(* IEC 61131-3 sources: SmartHomeNew/snapshots/2026-05-19 (part 2) *)

(* ---- GVL_STATE.gvl ---- *)
{attribute 'qualified_only'}
VAR_GLOBAL
    G_Floor_Temps : ARRAY[1..GVL_CONSTANTS.C_MAX_HEATING_CIRCUITS] OF REAL;
    G_Room_Temps : ARRAY[1..GVL_CONSTANTS.C_MAX_ZONES] OF REAL;
    G_Last_Valid_Room_Temps : ARRAY[1..GVL_CONSTANTS.C_MAX_ZONES] OF REAL;
    G_Last_Valid_Floor_Temps : ARRAY[1..GVL_CONSTANTS.C_MAX_HEATING_CIRCUITS] OF REAL;
    G_Temp_Sensor_Fault : ARRAY[1..GVL_CONSTANTS.C_MAX_ZONES] OF BOOL;
    G_Floor_Temp_Sensor_Fault : ARRAY[1..GVL_CONSTANTS.C_MAX_HEATING_CIRCUITS] OF BOOL;
    G_Room_Hum : ARRAY[1..GVL_CONSTANTS.C_MAX_ZONES] OF REAL;
    G_Room_CO2 : ARRAY[1..GVL_CONSTANTS.C_MAX_ZONES] OF REAL;
    G_Motion_Sensors : ARRAY[1..GVL_CONSTANTS.C_MAX_LIGHT_ZONES] OF BOOL;
    G_Door_Sensors : ARRAY[1..GVL_CONSTANTS.C_MAX_DOOR_SENSORS] OF BOOL;
    G_Window_Sensors : ARRAY[1..GVL_CONSTANTS.C_MAX_ZONES] OF BOOL;
    G_Water_Sensors : ARRAY[1..GVL_CONSTANTS.C_MAX_FLOOD_SENSORS] OF BOOL;
    G_Flood_Warning : ARRAY[1..GVL_CONSTANTS.C_MAX_FLOOD_SENSORS] OF BOOL;
    G_Flood_Alarm : ARRAY[1..GVL_CONSTANTS.C_MAX_FLOOD_SENSORS] OF BOOL;
    G_Flood_Warning_Rise : ARRAY[1..GVL_CONSTANTS.C_MAX_FLOOD_SENSORS] OF BOOL;
    G_Flood_Alarm_Rise : ARRAY[1..GVL_CONSTANTS.C_MAX_FLOOD_SENSORS] OF BOOL;
    G_Flood_Alarm_Fall : ARRAY[1..GVL_CONSTANTS.C_MAX_FLOOD_SENSORS] OF BOOL;
    G_Smoke_Sensors : ARRAY[1..GVL_CONSTANTS.C_MAX_SMOKE_SENSORS] OF BOOL;
    G_Methane_Sensors : ARRAY[1..GVL_CONSTANTS.C_MAX_METHANE_SENSORS] OF REAL;
    G_CO_Sensors : ARRAY[1..GVL_CONSTANTS.C_MAX_CO_SENSORS] OF REAL;
    G_Manifold_Pressures : ARRAY[1..GVL_CONSTANTS.C_MAX_MANIFOLDS] OF REAL;
    G_Manifold_Currents : ARRAY[1..GVL_CONSTANTS.C_MAX_MANIFOLDS] OF REAL;
    G_Predictive_Pump_Pressure_Drop : ARRAY[1..GVL_CONSTANTS.C_MAX_MANIFOLDS] OF BOOL;
    G_Predictive_Pump_Current_Rise : ARRAY[1..GVL_CONSTANTS.C_MAX_MANIFOLDS] OF BOOL;
    G_Manifold_T_Supply : ARRAY[1..GVL_CONSTANTS.C_MAX_MANIFOLDS] OF REAL;
    G_Manifold_T_Return : ARRAY[1..GVL_CONSTANTS.C_MAX_MANIFOLDS] OF REAL;
    G_Boiler_Flame : ARRAY[1..GVL_CONSTANTS.C_MAX_BOILERS] OF BOOL;
    G_Boiler_Error : ARRAY[1..GVL_CONSTANTS.C_MAX_BOILERS] OF BOOL;
    G_Boiler_OT_Online : ARRAY[1..GVL_CONSTANTS.C_MAX_BOILERS] OF BOOL;
    G_Boiler_OT_Command_Ack : ARRAY[1..GVL_CONSTANTS.C_MAX_BOILERS] OF BOOL;
    G_Boiler_OT_Command_Timeout : ARRAY[1..GVL_CONSTANTS.C_MAX_BOILERS] OF BOOL;
    G_Boiler_OT_Heartbeat_Timeout : ARRAY[1..GVL_CONSTANTS.C_MAX_BOILERS] OF BOOL;
    G_Boiler_OT_Adapter_Error : ARRAY[1..GVL_CONSTANTS.C_MAX_BOILERS] OF BOOL;
    G_Boiler_OT_Heartbeat_Age_MS : ARRAY[1..GVL_CONSTANTS.C_MAX_BOILERS] OF UDINT;
    G_Boiler_OT_Command_Age_MS : ARRAY[1..GVL_CONSTANTS.C_MAX_BOILERS] OF UDINT;
    G_Boiler_OT_Adapter_State : ARRAY[1..GVL_CONSTANTS.C_MAX_BOILERS] OF E_OpenTherm_Adapter_State;
    G_Boiler_OT_Error_State : ARRAY[1..GVL_CONSTANTS.C_MAX_BOILERS] OF E_OpenTherm_Error;
    G_Boiler_OT_Enable : ARRAY[1..GVL_CONSTANTS.C_MAX_BOILERS] OF BOOL;
    G_Boiler_OT_Setpoint : ARRAY[1..GVL_CONSTANTS.C_MAX_BOILERS] OF REAL;
    G_Heating_Cascade_Available : BOOL;
    G_Heating_Cascade_Degraded : BOOL;
    G_Heating_Cascade_Partial_Capacity : BOOL;
    G_Heating_Cascade_No_Flame : BOOL;
    G_Heating_Cascade_Transport_Degraded : BOOL;
    G_Heating_Cascade_Ignition_Timeout : BOOL;
    G_Heating_Cascade_Active_Boilers : UINT;
    G_Heating_Cascade_Available_Boilers : UINT;
    G_Physical_Switches : ARRAY[1..GVL_CONSTANTS.C_MAX_LIGHT_ZONES] OF BOOL;
    G_Socket_Switches : ARRAY[1..GVL_CONSTANTS.C_MAX_SOCKETS] OF BOOL;
    G_Outdoor_Temp : REAL;
    G_Supply_Temps : ARRAY[1..GVL_CONSTANTS.C_MAX_SUPPLY_TEMPS] OF REAL;
    G_DHW_Temp : REAL;
    G_DHW_Pressure : REAL;
    G_Zone_Valves : ARRAY[1..GVL_CONSTANTS.C_MAX_HEATING_CIRCUITS] OF BOOL;
    G_Manifold_Pumps : ARRAY[1..GVL_CONSTANTS.C_MAX_MANIFOLDS] OF BOOL;
    G_Manifold_Valves : ARRAY[1..GVL_CONSTANTS.C_MAX_MANIFOLDS] OF REAL;
    G_Manifold_End_Switches : ARRAY[1..GVL_CONSTANTS.C_MAX_MANIFOLDS] OF BOOL;
    G_Supply_Fans : ARRAY[1..GVL_CONSTANTS.C_MAX_SUPPLY_FANS] OF REAL;
    G_Exhaust_Fans : ARRAY[1..GVL_CONSTANTS.C_MAX_EXHAUST_FANS] OF REAL;
    G_Vent_Heater_Power : ARRAY[1..GVL_CONSTANTS.C_MAX_BOILERS] OF REAL;
    G_Lighting_Levels : ARRAY[1..GVL_CONSTANTS.C_MAX_LIGHT_ZONES] OF BYTE;
    G_Blinds_Positions : ARRAY[1..GVL_CONSTANTS.C_MAX_BLINDS] OF BYTE;
    G_Socket_States : ARRAY[1..GVL_CONSTANTS.C_MAX_SOCKETS] OF BOOL;
    G_DHW_Heating_Pump : BOOL;
    G_DHW_Circ_Pump : BOOL;
    G_Backup_Circulation_Pump : BOOL;
    G_Electric_Heater_Enable : BOOL;
    G_Safety_Gas_Alarm : BOOL;
    G_Safety_Leak_Alarm : BOOL;
    G_Safety_Smoke_Alarm : BOOL;
    G_Safety_Emergency_Stop : BOOL;
    G_Safety_Gas_Latched : BOOL;
    G_Safety_Leak_Latched : BOOL;
    G_Safety_Smoke_Latched : BOOL;
    G_Safety_Freeze_Risk : BOOL;
    G_System_Mode : E_System_Operating_Mode := E_System_Operating_Mode.MODE_NORMAL;
    G_System_Mode_Text : STRING(64);
    G_Heating_IO_Fault : BOOL;
    G_Heating_Sensor_Fault : BOOL;
    G_Heating_Subsystem_Degraded : BOOL;
    G_Allocation_Policy_Active : BOOL;
    G_Allocation_Freeze_Bypass_Active : BOOL;
    G_Allocation_DHW_Bypass_Active : BOOL;
    G_Allocation_Budget_Max : REAL;
    G_Allocation_Budget_Used : REAL;
    G_Allocation_Requested : ARRAY[1..GVL_CONSTANTS.C_MAX_MANIFOLDS] OF BOOL;
    G_Allocation_Allowed : ARRAY[1..GVL_CONSTANTS.C_MAX_MANIFOLDS] OF BOOL;
    G_Allocation_Filtered : ARRAY[1..GVL_CONSTANTS.C_MAX_MANIFOLDS] OF BOOL;
    G_Allocation_Block_Reason : ARRAY[1..GVL_CONSTANTS.C_MAX_MANIFOLDS] OF E_Heating_Allocation_Block_Reason;
    G_Allocation_Effective_Priority : ARRAY[1..GVL_CONSTANTS.C_MAX_MANIFOLDS] OF INT;
    G_Policy_Target_Adjustment_Active : BOOL;
    G_Policy_Target_Adjustment_Applied : REAL;
    G_Policy_Priority_Multiplier_Applied : REAL;
    G_Policy_Priority_Bridge_Active : BOOL;
    G_Policy_Priority_Bias_Applied : ARRAY[1..GVL_CONSTANTS.C_MAX_MANIFOLDS] OF REAL;
    G_Policy_Priority_Effective : ARRAY[1..GVL_CONSTANTS.C_MAX_MANIFOLDS] OF INT;
    G_Heating_RootCause : E_Heating_RootCause := E_Heating_RootCause.RC_NONE;
    G_Heating_RootConfidence : REAL;
    G_Heating_Confidence : REAL := 1.0;
    G_Heating_Error_Score : REAL := 0.0;
    G_Heating_Confidence_Reason_Code : INT := 0;
    G_Heating_Confidence_Reason_Text : STRING(128) := 'OK';
    G_DHW_IO_Fault : BOOL;
    G_DHW_Sensor_Fault : BOOL;
    G_DHW_Subsystem_Degraded : BOOL;
    G_Ventilation_IO_Fault : BOOL;
    G_Ventilation_Subsystem_Degraded : BOOL;
    G_Lighting_IO_Fault : BOOL;
    G_Lighting_Subsystem_Degraded : BOOL;
    G_Access_Comm_Fault : BOOL;
    G_Evacuation_Lighting_Active : BOOL;
    G_Evac_Hazard_Zone : ARRAY[1..GVL_CONSTANTS.C_MAX_LIGHT_ZONES] OF BOOL;
    G_Evac_Guidance : ARRAY[1..GVL_CONSTANTS.C_MAX_LIGHT_ZONES] OF INT;
    G_Rule_Actions : ARRAY[1..GVL_CONSTANTS.C_MAX_RULES] OF ST_Rule_Action;
    G_Sim_Lights : ARRAY[1..GVL_CONSTANTS.C_MAX_LIGHT_ZONES] OF BOOL;
    G_Freeze_Hardware_Degraded : BOOL;
    G_Freeze_Hardware_Failed : BOOL;
    G_Water_Zone_Enable : ARRAY[1..GVL_CONSTANTS.C_MAX_WATER_ZONES] OF BOOL;
    G_Water_Zone_Open_FB : ARRAY[1..GVL_CONSTANTS.C_MAX_WATER_ZONES] OF BOOL;
    G_Water_Zone_Close_FB : ARRAY[1..GVL_CONSTANTS.C_MAX_WATER_ZONES] OF BOOL;
    G_Water_Zone_Exercise_Active : ARRAY[1..GVL_CONSTANTS.C_MAX_WATER_ZONES] OF BOOL;
    G_Preheat_Request : BOOL;
    G_Freeze_Request : BOOL;
    G_Target_Temperature : REAL;
END_VAR

(* ---- GVL_SYSTEM_COORDINATION.gvl ---- *)
{attribute 'qualified_only'}
VAR_GLOBAL
    G_System_Degraded : BOOL := FALSE;

    G_Block_Heating : BOOL := FALSE;
    G_Block_Ventilation : BOOL := FALSE;
    G_Block_Lighting_Override : BOOL := FALSE;
    G_Block_Sockets_Override : BOOL := FALSE;

    G_Coordination_Code : UDINT := 0;
    G_Coordination_Status_Msg : STRING(200) := '';
END_VAR

(* ---- GVL_TEMPORAL_CAUSALITY_CLOSURE_FABRIC.gvl ---- *)
VAR_GLOBAL
    Temporal_Causality_Closure_Valid : BOOL := FALSE;
    Temporal_Causality_Closure_Granted : BOOL := FALSE;

    Temporal_Causality_Coherent : BOOL := FALSE;
    Monotonic_Reality_Timeline_Valid : BOOL := FALSE;
    Distributed_Temporal_Alignment_Stable : BOOL := FALSE;
    Recovery_Revocation_Ordering_Valid : BOOL := FALSE;

    Temporal_Causality_Lineage_Coherent : BOOL := FALSE;
    Distributed_Temporal_Consensus_Valid : BOOL := FALSE;

    Temporal_Fork_Detected : BOOL := FALSE;
    Stale_Causality_Application_Detected : BOOL := FALSE;
    Recovery_Before_Revocation_Detected : BOOL := FALSE;
    Distributed_Timeline_Drift_Detected : BOOL := FALSE;

    Temporal_Causality_Epoch : UDINT := 0;
END_VAR

(* ---- GVL_TEST_PANEL_RESULT.gvl ---- *)
{attribute 'qualified_only'}
VAR_GLOBAL
    // === RESULT VIEW ONLY ===
    G_Enable : BOOL := FALSE;
    G_Scenario_ID : INT := 0;
    G_Scenario_Run : BOOL := FALSE;
    G_Scenario_Active : BOOL := FALSE;

    G_Test_Result_Line : STRING(200) := 'Idle';
    G_Result_Passed : BOOL := FALSE;
    G_Result_Status_Msg : STRING(200) := 'Idle';
    G_Result_Fail_Code : UDINT := 0;

    G_Result_Base_Priority : INT := 0;
    G_Result_Expected_Adjusted_Priority : INT := 0;
    G_Result_Actual_Adjusted_Priority : INT := 0;
    G_Result_Delta : INT := 0;

    G_Result_Budget_Exceeded : BOOL := FALSE;
    G_Result_Used_Thermal_Budget : REAL := 0.0;
    G_Result_Manifold_Enabled : ARRAY[1..GVL_CONSTANTS.C_MAX_MANIFOLDS] OF BOOL;
END_VAR

(* ---- GVL_Water_Isolation_Authority.gvl ---- *)
{attribute 'qualified_only'}
VAR_GLOBAL
    // ==============================================================================
    // Water/Flood authority arbitration publication.
    // ==============================================================================
    //
    // Explicit deterministic authority decision layer.
    //
    // This layer:
    // - evaluates selective isolation authority;
    // - preserves conservative global fallback;
    // - publishes explainable authority decisions.
    //
    // This layer does NOT directly own physical outputs.
    // ==============================================================================

    G_Authority_State : ARRAY[1..GVL_CONSTANTS.C_MAX_FLOOD_SENSORS] OF ST_Water_Isolation_Authority_State;

    // Aggregated authority visibility.
    G_Any_Selective_Authority_Allowed : BOOL;
    G_Any_Global_Fallback_Required : BOOL;
    G_Any_Authority_Denied : BOOL;

    // Runtime lifecycle.
    G_Authority_Valid : BOOL;
    G_Last_Update_MS : UDINT;

    // Explainability.
    G_Status_Code : UINT;
    G_Status_Text : STRING(128);
END_VAR

(* ---- GVL_Water_Output_Reconciliation.gvl ---- *)
{attribute 'qualified_only'}
VAR_GLOBAL
    G_Reconciliation_State : ARRAY[1..64] OF ST_Water_Output_Reconciliation_State;

    G_Any_Runtime_Mismatch : BOOL;
    G_Any_Confirmation_Mismatch : BOOL;
    G_Any_Conflict_Detected : BOOL;

    G_Runtime_Valid : BOOL;
    G_Last_Update_MS : UDINT;

    G_Status_Code : UINT;
    G_Status_Text : STRING(128);
END_VAR

(* ---- GVL_Water_Recovery_Runtime.gvl ---- *)
{attribute 'qualified_only'}
VAR_GLOBAL
    G_Recovery_State : ARRAY[1..64] OF ST_Water_Recovery_Runtime_State;

    G_Any_Recovery_Denied : BOOL;
    G_Any_Unsafe_Recovery : BOOL;

    G_Runtime_Valid : BOOL;
    G_Last_Update_MS : UDINT;

    G_Status_Code : UINT;
    G_Status_Text : STRING(128);
END_VAR

(* ---- GVL_Water_Runtime_Projection.gvl ---- *)
{attribute 'qualified_only'}
VAR_GLOBAL
    // ==============================================================================
    // Canonical Water/Flood runtime projection publication surface.
    // ==============================================================================
    //
    // Observe/publish-only semantic boundary.
    //
    // This GVL is intended to become the canonical semantic transfer layer
    // between:
    //
    // - leak detection/runtime execution;
    // - safety governance;
    // - future selective isolation semantics;
    // - observability/explainability;
    // - supervisory publication.
    //
    // This GVL does NOT:
    // - own outputs;
    // - own valve authority;
    // - directly close/open valves;
    // - override runtime.
    //
    // Canonical topology direction:
    //
    // physical input
    //   -> normalized leak semantics
    //   -> logical leak sensor
    //   -> hydraulic mapping
    //   -> isolation semantics
    //   -> governance/arbitration
    //   -> output projection
    //   -> observability/publication
    // ==============================================================================

    G_Leak_Runtime_State : ARRAY[1..GVL_CONSTANTS.C_MAX_FLOOD_SENSORS] OF ST_Water_Leak_Runtime_State;

    // Projection lifecycle.
    G_Projection_Valid : BOOL;
    G_Last_Projection_MS : UDINT;

    // Active runtime compatibility visibility.
    G_Global_Leak_Active : BOOL;
    G_Global_Warning_Active : BOOL;

    // Observability contract.
    G_Runtime_Projection_Status_Code : UINT;
    G_Runtime_Projection_Status_Text : STRING(128);
END_VAR

(* ---- GVL_Water_Topology_Validation.gvl ---- *)
{attribute 'qualified_only'}
VAR_GLOBAL
    G_Validation_State : ARRAY[1..64] OF ST_Water_Topology_Validation_State;

    G_Any_Invalid : BOOL;
    G_Any_Ambiguous : BOOL;
    G_Any_Global_Fallback_Required : BOOL;

    G_Runtime_Valid : BOOL;
    G_Last_Update_MS : UDINT;

    G_Status_Code : UINT;
    G_Status_Text : STRING(128);
END_VAR

(* ---- GVL_Water_Valve_Feedback.gvl ---- *)
{attribute 'qualified_only'}
VAR_GLOBAL
    G_Valve_Feedback_State : ARRAY[1..64] OF ST_Water_Valve_Feedback_State;

    G_Any_Degraded : BOOL;
    G_Any_Timeout : BOOL;
    G_Any_Conflict : BOOL;

    G_Runtime_Valid : BOOL;
    G_Last_Update_MS : UDINT;

    G_Status_Code : UINT;
    G_Status_Text : STRING(128);
END_VAR

(* ---- FB_Access_Output_Projection.st ---- *)
FUNCTION_BLOCK FB_Access_Output_Projection
VAR_INPUT
    VI_Lock_1_Open : BOOL;
    VI_Lock_1_Close : BOOL;
    VI_Lock_2_Open : BOOL;
    VI_Lock_2_Close : BOOL;
    VI_Gate_Open : BOOL;
    VI_Wicket_Open : BOOL;
END_VAR

GVL_ACCESS_OUTPUT.DO_Lock_1_Open := VI_Lock_1_Open;
GVL_ACCESS_OUTPUT.DO_Lock_1_Close := VI_Lock_1_Close;
GVL_ACCESS_OUTPUT.DO_Lock_2_Open := VI_Lock_2_Open;
GVL_ACCESS_OUTPUT.DO_Lock_2_Close := VI_Lock_2_Close;
GVL_ACCESS_OUTPUT.DO_Gate_Open := VI_Gate_Open;
GVL_ACCESS_OUTPUT.DO_Wicket_Open := VI_Wicket_Open;

END_FUNCTION_BLOCK
// >>> BULK_SYNC_ANCHOR: FB_Access_Output_Projection <<<

(* ---- FB_ADS_Runtime_Adapter.st ---- *)
FUNCTION_BLOCK FB_ADS_Runtime_Adapter
VAR_INPUT
    VI_Enable : BOOL;
    VI_System_Time_MS : UDINT;
END_VAR
VAR
    L_Frame : ST_Runtime_Bus_Frame;
    L_TX_Index : UINT;
END_VAR

IF NOT VI_Enable THEN
    RETURN;
END_IF;

L_TX_Index := UDINT_TO_UINT(GVL_Runtime_Bus.G_Last_Sequence_Id);

IF (L_TX_Index >= 1)
   AND (L_TX_Index <= 128) THEN

    L_Frame := GVL_Runtime_Bus.G_TX_Frames[L_TX_Index];

    IF L_Frame.Frame_Valid THEN

        IF GVL_Distributed_Authority.G_Distributed_Safety_Barrier_OK
           AND GVL_Runtime_Sessions.G_Runtime_Valid
           AND NOT GVL_Runtime_Sessions.G_Any_Stale_Session
           AND NOT GVL_Runtime_Sessions.G_Any_Quarantined_Session THEN

            L_Frame.Frame_Ack_Received := TRUE;
            L_Frame.Replication_Consistent := TRUE;
            L_Frame.Replication_Rejected := FALSE;
            L_Frame.Status_Code := 0;

        ELSE

            L_Frame.Frame_Ack_Received := FALSE;
            L_Frame.Replication_Consistent := FALSE;
            L_Frame.Replication_Rejected := TRUE;
            L_Frame.Status_Code := 2;

        END_IF;

        GVL_Runtime_Bus.G_TX_Frames[L_TX_Index] := L_Frame;
        GVL_Runtime_Bus.G_TX_Healthy := L_Frame.Replication_Consistent;
        GVL_Runtime_Bus.G_Any_Replication_Rejected := L_Frame.Replication_Rejected;

    END_IF;

END_IF;

END_FUNCTION_BLOCK

(* ---- FB_Behavior_Adapt.st ---- *)
FUNCTION_BLOCK FB_Behavior_Adapt
VAR_INPUT
    iScenario : E_System_Reason_Code;
    iSuccess : BOOL;
    iMeasuredValue : REAL;
    iZone : INT;
    iConfidence : REAL;
END_VAR

VAR
    L_Stats : ST_Scenario_Stats;
    L_Zone : ST_Zone_Adapt_State;
    L_Adjustment : REAL;
    L_Decay : REAL;
    idx : INT;
END_VAR

IF NOT GVL_BEHAVIOR_ADAPT.G_Adapt_Enabled THEN RETURN; END_IF;

idx := USINT_TO_INT(iScenario);

L_Stats := GVL_BEHAVIOR_ADAPT.G_Scenario_Stats[idx];
L_Stats.Activations := L_Stats.Activations + 1;

IF iSuccess THEN
    L_Stats.Success_Count := L_Stats.Success_Count + 1;
ELSE
    L_Stats.Failure_Count := L_Stats.Failure_Count + 1;
END_IF;

IF L_Stats.Activations > 0 THEN
    L_Stats.Success_Rate := UDINT_TO_REAL(L_Stats.Success_Count) / UDINT_TO_REAL(L_Stats.Activations);
END_IF;

IF (iScenario = REASON_SCENARIO_VENT_BOOST) AND (iZone >= 1) AND (iZone <= GVL_CONSTANTS.C_MAX_ZONES) THEN

    L_Zone := GVL_BEHAVIOR_ADAPT.G_VentBoost_Zone_Adapt[iZone];

    IF L_Zone.Zone_Weight = 0.0 THEN
        L_Zone.Zone_Weight := GVL_BEHAVIOR_ADAPT.G_Adapt_Default_Zone_Weight;
    END_IF;

    L_Decay := GVL_BEHAVIOR_ADAPT.G_Decay_Factor;
    L_Zone.Zone_Weight := L_Zone.Zone_Weight * L_Decay;
    L_Zone.Confidence := L_Zone.Confidence * L_Decay;

    L_Zone.Activations := L_Zone.Activations + 1;

    IF iSuccess THEN
        L_Zone.Success_Count := L_Zone.Success_Count + 1;
    ELSE
        L_Zone.Failure_Count := L_Zone.Failure_Count + 1;
    END_IF;

    IF L_Zone.Activations > 0 THEN
        L_Zone.Success_Rate := UDINT_TO_REAL(L_Zone.Success_Count) / UDINT_TO_REAL(L_Zone.Activations);
    END_IF;

    IF iConfidence >= GVL_BEHAVIOR_ADAPT.G_Adapt_Min_Confidence THEN
        L_Zone.Confidence := L_Zone.Confidence +
            (iConfidence - L_Zone.Confidence) * GVL_BEHAVIOR_ADAPT.G_Confidence_Learning_Rate;
    END_IF;

    IF (GVL_BEHAVIOR_ADAPT.G_Adapt_Update_Threshold > 0) AND
       ((L_Zone.Activations MOD INT_TO_UDINT(GVL_BEHAVIOR_ADAPT.G_Adapt_Update_Threshold)) = 0) THEN

        L_Adjustment :=
            (L_Zone.Success_Rate - 0.5)
            * GVL_BEHAVIOR_ADAPT.G_Adapt_Learning_Rate
            * L_Zone.Confidence;

        L_Zone.Zone_Weight := LIMIT(0.5, L_Zone.Zone_Weight + L_Adjustment, 2.0);

    END_IF;

    L_Zone.Last_Update_MS := GVL_TIME_SERVICE.G_Now_MS;

    GVL_BEHAVIOR_ADAPT.G_VentBoost_Zone_Adapt[iZone] := L_Zone;

END_IF;

GVL_BEHAVIOR_ADAPT.G_Scenario_Stats[idx] := L_Stats;
END_FUNCTION_BLOCK

(* ---- FB_Boiler_Cascade_Manager.st ---- *)
FUNCTION_BLOCK FB_Boiler_Cascade_Manager
VAR_INPUT
    VI_Enable : BOOL;
    VI_System_Time_MS : UDINT;
    VI_Boiler_Stop : BOOL;

    VI_DHW_Heating_Demand : BOOL;
    VI_DHW_Target_Temp : REAL;

    VI_Target_Supply_Temp : REAL;
    VI_Demand_Power : REAL; // 0..500% (сумма запросов от 5 смесительных узлов)

    VI_Boiler_Flame_Status : ARRAY[1..GVL_CONSTANTS.C_MAX_BOILERS] OF BOOL;
    VI_Boiler_Error_Status : ARRAY[1..GVL_CONSTANTS.C_MAX_BOILERS] OF BOOL;
    VI_Boiler_OT_Online : ARRAY[1..GVL_CONSTANTS.C_MAX_BOILERS] OF BOOL;
    VI_Boiler_Modulation : ARRAY[1..GVL_CONSTANTS.C_MAX_BOILERS] OF REAL;
END_VAR

VAR_OUTPUT
    VO_Boiler_Enable : ARRAY[1..GVL_CONSTANTS.C_MAX_BOILERS] OF BOOL;
    VO_Boiler_Setpoint : ARRAY[1..GVL_CONSTANTS.C_MAX_BOILERS] OF REAL;
    VO_Lead_Boiler : BYTE;
END_VAR

VAR
    L_i : INT;
    L_Lead_Boiler : BYTE := 1;

    L_Last_Rotation_MS : UDINT := 0;
    L_Rotation_Initialized : BOOL := FALSE;
    L_Rotation_Period_MS : UDINT := 604800000; // 168h

    L_Lead_Available : BOOL;
    L_Reserve_Available : BOOL;
    L_Reserve_Boiler : BYTE;
    L_Start_Reserve : BOOL;
    L_Target_Setpoint : REAL;
    L_Flame_Miss_Timer : ARRAY[1..GVL_CONSTANTS.C_MAX_BOILERS] OF TON;
END_VAR

// Сброс выходов по умолчанию
FOR L_i := 1 TO GVL_CONSTANTS.C_MAX_BOILERS DO
    VO_Boiler_Enable[L_i] := FALSE;
    VO_Boiler_Setpoint[L_i] := 0.0;
END_FOR;

// Инициализация ротации
IF NOT L_Rotation_Initialized THEN
    L_Last_Rotation_MS := VI_System_Time_MS;
    L_Rotation_Initialized := TRUE;
END_IF;

// Принудительная остановка
IF VI_Boiler_Stop THEN
    VO_Lead_Boiler := L_Lead_Boiler;
    RETURN;
END_IF;

// Ротация строго каждые 168 часов
IF (VI_System_Time_MS - L_Last_Rotation_MS) >= L_Rotation_Period_MS THEN
    IF GVL_CONSTANTS.C_MAX_BOILERS > 1 THEN
        L_Lead_Boiler := 3 - L_Lead_Boiler;
    END_IF;
    L_Last_Rotation_MS := VI_System_Time_MS;
END_IF;

L_Reserve_Boiler := SEL(L_Lead_Boiler = 1, 1, 2);

L_Lead_Available :=
    VI_Boiler_OT_Online[L_Lead_Boiler] AND
    NOT VI_Boiler_Error_Status[L_Lead_Boiler];

L_Reserve_Available :=
    (GVL_CONSTANTS.C_MAX_BOILERS > 1) AND
    VI_Boiler_OT_Online[L_Reserve_Boiler] AND
    NOT VI_Boiler_Error_Status[L_Reserve_Boiler];

// Контроль "команда есть, пламени нет" для ведущего котла
L_Flame_Miss_Timer[L_Lead_Boiler](
    IN := VI_Enable AND L_Lead_Available AND NOT VI_DHW_Heating_Demand AND NOT VI_Boiler_Flame_Status[L_Lead_Boiler],
    PT := T#120s
);

IF L_Flame_Miss_Timer[L_Lead_Boiler].Q AND L_Reserve_Available THEN
    L_Lead_Boiler := L_Reserve_Boiler;
    L_Last_Rotation_MS := VI_System_Time_MS;
    L_Lead_Available :=
        VI_Boiler_OT_Online[L_Lead_Boiler] AND
        NOT VI_Boiler_Error_Status[L_Lead_Boiler];
    L_Reserve_Boiler := SEL(L_Lead_Boiler = 1, 1, 2);
    L_Reserve_Available :=
        (GVL_CONSTANTS.C_MAX_BOILERS > 1) AND
        VI_Boiler_OT_Online[L_Reserve_Boiler] AND
        NOT VI_Boiler_Error_Status[L_Reserve_Boiler];
END_IF;

// Нет запроса тепла
IF NOT VI_Enable THEN
    VO_Lead_Boiler := L_Lead_Boiler;
    RETURN;
END_IF;

// Целевая уставка
IF VI_DHW_Heating_Demand THEN
    L_Target_Setpoint := LIMIT(20.0, VI_DHW_Target_Temp + 15.0, 85.0);
ELSE
    L_Target_Setpoint := LIMIT(20.0, VI_Target_Supply_Temp + 5.0, 80.0);
END_IF;

// Выбор ведущего по доступности
IF NOT L_Lead_Available AND L_Reserve_Available THEN
    L_Lead_Boiler := L_Reserve_Boiler;
    L_Lead_Available := TRUE;
    L_Reserve_Boiler := SEL(L_Lead_Boiler = 1, 1, 2);
    L_Reserve_Available :=
        (GVL_CONSTANTS.C_MAX_BOILERS > 1) AND
        VI_Boiler_OT_Online[L_Reserve_Boiler] AND
        NOT VI_Boiler_Error_Status[L_Reserve_Boiler];
END_IF;

// Основной котёл
IF L_Lead_Available THEN
    VO_Boiler_Enable[L_Lead_Boiler] := TRUE;
    VO_Boiler_Setpoint[L_Lead_Boiler] := L_Target_Setpoint;
END_IF;

// Резервный котёл: >80% или отказ основного
L_Start_Reserve :=
    L_Reserve_Available AND
    (
        (VI_Demand_Power > 80.0) OR
        (NOT L_Lead_Available)
    );

IF L_Start_Reserve THEN
    VO_Boiler_Enable[L_Reserve_Boiler] := TRUE;
    VO_Boiler_Setpoint[L_Reserve_Boiler] := L_Target_Setpoint;
END_IF;

VO_Lead_Boiler := L_Lead_Boiler;
END_FUNCTION_BLOCK

(* ---- FB_Boiler_OpenTherm_Interface.st ---- *)
FUNCTION_BLOCK FB_Boiler_OpenTherm_Interface
VAR_INPUT
    VI_Enable : ARRAY[1..GVL_CONSTANTS.C_MAX_BOILERS] OF BOOL;
    VI_Setpoint : ARRAY[1..GVL_CONSTANTS.C_MAX_BOILERS] OF REAL;

    VI_OT_Online : ARRAY[1..GVL_CONSTANTS.C_MAX_BOILERS] OF BOOL;
    VI_OT_Error : ARRAY[1..GVL_CONSTANTS.C_MAX_BOILERS] OF BOOL;
END_VAR

VAR_OUTPUT
    VO_OT_Enable : ARRAY[1..GVL_CONSTANTS.C_MAX_BOILERS] OF BOOL;
    VO_OT_Setpoint : ARRAY[1..GVL_CONSTANTS.C_MAX_BOILERS] OF REAL;
    VO_OT_Command_Valid : ARRAY[1..GVL_CONSTANTS.C_MAX_BOILERS] OF BOOL;
END_VAR

VAR
    L_i : INT;
    L_Setpoint : REAL;
    L_Setpoint_x10 : UINT;
    L_Command_Enable : BOOL;
    L_Command_Changed : BOOL;
    L_Last_Command_Enable : ARRAY[1..GVL_CONSTANTS.C_MAX_BOILERS] OF BOOL;
    L_Last_Command_Setpoint_x10 : ARRAY[1..GVL_CONSTANTS.C_MAX_BOILERS] OF UINT;
END_VAR

FOR L_i := 1 TO GVL_CONSTANTS.C_MAX_BOILERS DO

    VO_OT_Enable[L_i] := FALSE;
    VO_OT_Setpoint[L_i] := 0.0;
    VO_OT_Command_Valid[L_i] := FALSE;

    L_Command_Enable := FALSE;
    L_Setpoint := 0.0;
    L_Setpoint_x10 := 0;

    // ======================================================
    // COMMAND VALIDATION
    // ======================================================
    IF VI_Enable[L_i] AND VI_OT_Online[L_i] AND NOT VI_OT_Error[L_i] THEN
        L_Command_Enable := TRUE;
        L_Setpoint := LIMIT(20.0, VI_Setpoint[L_i], 80.0);
        L_Setpoint_x10 := REAL_TO_UINT(L_Setpoint * 10.0);

        VO_OT_Enable[L_i] := TRUE;
        VO_OT_Setpoint[L_i] := L_Setpoint;
    END_IF;

    // ======================================================
    // PHYSICAL ADAPTER COMMAND IMAGE
    // ======================================================
    GVL_OPENTHERM_ADAPTER.G_Command[L_i].Enable := L_Command_Enable;
    GVL_OPENTHERM_ADAPTER.G_Command[L_i].Setpoint_x10 := L_Setpoint_x10;

    // Sequence is advanced only when the actual command image changes.
    // This keeps the command stable long enough for adapter ACK validation.
    L_Command_Changed :=
        (L_Command_Enable <> L_Last_Command_Enable[L_i]) OR
        (L_Setpoint_x10 <> L_Last_Command_Setpoint_x10[L_i]);

    IF L_Command_Changed THEN
        GVL_OPENTHERM_ADAPTER.G_Command[L_i].Sequence :=
            GVL_OPENTHERM_ADAPTER.G_Command[L_i].Sequence + 1;

        GVL_OPENTHERM_ADAPTER.G_Command[L_i].Last_Write_MS :=
            GVL_STATUS.G_System_Time_MS;

        L_Last_Command_Enable[L_i] := L_Command_Enable;
        L_Last_Command_Setpoint_x10[L_i] := L_Setpoint_x10;
    END_IF;

    // Command is valid only when the adapter confirms the current stable sequence.
    VO_OT_Command_Valid[L_i] :=
        L_Command_Enable AND
        GVL_OPENTHERM_ADAPTER.G_Status[L_i].Command_Ack AND
        (NOT GVL_OPENTHERM_ADAPTER.G_Status[L_i].Adapter_Error) AND
        GVL_OPENTHERM_ADAPTER.G_Status[L_i].Adapter_Online;

END_FOR;

END_FUNCTION_BLOCK

(* ---- FB_Cluster_Runtime_FSM.st ---- *)
FUNCTION_BLOCK FB_Cluster_Runtime_FSM
VAR_INPUT
    VI_Enable : BOOL;
    VI_System_Time_MS : UDINT;
END_VAR
VAR
    L_Finalized_Runtime_Continuity : BOOL;
END_VAR

IF NOT VI_Enable THEN
    GVL_Cluster_Runtime_FSM.G_Runtime_Valid := FALSE;
    RETURN;
END_IF;

// Finalized runtime continuity proof chain.
L_Finalized_Runtime_Continuity :=
    GVL_SEMANTIC_PROGRESS.Semantic_Forward_Progress_Valid
    AND GVL_SEMANTIC_PROGRESS.Semantic_Execution_Continuity_OK
    AND NOT GVL_SEMANTIC_PROGRESS.Semantic_Progress_Lease_Expired
    AND NOT GVL_SEMANTIC_PROGRESS.Semantic_Progress_Quarantine_Active
    AND GVL_RUNTIME_SNAPSHOT.Snapshot_Frozen
    AND GVL_RUNTIME_SNAPSHOT.Snapshot_Publication_Allowed
    AND GVL_RUNTIME_SNAPSHOT.Snapshot_Copy_Valid
    AND GVL_RUNTIME_SNAPSHOT.Snapshot_Isolation_Valid
    AND NOT GVL_RUNTIME_SNAPSHOT.Snapshot_Mutation_Detected
    AND GVL_DISTRIBUTED_SNAPSHOT.Distributed_Publication_Reconciled
    AND GVL_DISTRIBUTED_SNAPSHOT.Distributed_Publication_Freeze_Valid
    AND GVL_DISTRIBUTED_SNAPSHOT.Distributed_Snapshot_Consistent
    AND GVL_DISTRIBUTED_COMMIT.Distributed_Commit_Valid
    AND GVL_DISTRIBUTED_COMMIT.Publication_Prepare_Valid
    AND GVL_DISTRIBUTED_COMMIT.Publication_Commit_Confirmed
    AND NOT GVL_DISTRIBUTED_COMMIT.Peer_Commit_Mismatch
    AND NOT GVL_DISTRIBUTED_COMMIT.Commit_Lease_Expired
    AND GVL_OUTPUT_EPOCH.Output_Publication_Valid
    AND GVL_OUTPUT_EPOCH.Output_Runtime_Epoch_Valid
    AND NOT GVL_OUTPUT_EPOCH.Output_Lease_Expired
    AND NOT GVL_OUTPUT_EPOCH.Output_Forced_Safe_Decay
    AND GVL_COMMAND_VERIFY.PreOutput_Barrier_OK
    AND NOT GVL_COMMAND_VERIFY.PreOutput_Block_IO;

// Reset runtime states.
GVL_Cluster_Runtime_FSM.G_State_Startup := FALSE;
GVL_Cluster_Runtime_FSM.G_State_Discovery := FALSE;
GVL_Cluster_Runtime_FSM.G_State_Synchronization := FALSE;
GVL_Cluster_Runtime_FSM.G_State_Operational := FALSE;
GVL_Cluster_Runtime_FSM.G_State_Degraded := FALSE;
GVL_Cluster_Runtime_FSM.G_State_Observer_Only := FALSE;
GVL_Cluster_Runtime_FSM.G_State_Recovery_Lock := FALSE;
GVL_Cluster_Runtime_FSM.G_State_Quarantine := FALSE;

// Startup state.
IF NOT GVL_Distributed_Runtime.G_Runtime_Valid THEN

    GVL_Cluster_Runtime_FSM.G_State_Startup := TRUE;

    GVL_Cluster_Runtime_FSM.G_Status_Code := 1;
    GVL_Cluster_Runtime_FSM.G_Status_Text :=
        'Cluster runtime startup';

ELSIF GVL_Runtime_Discovery.G_Runtime_Valid
   AND NOT GVL_Runtime_Discovery.G_Any_Discovery_Rejected THEN

    GVL_Cluster_Runtime_FSM.G_State_Discovery := TRUE;

    GVL_Cluster_Runtime_FSM.G_Status_Code := 2;
    GVL_Cluster_Runtime_FSM.G_Status_Text :=
        'Cluster runtime discovery';

END_IF;

// Synchronization state.
IF GVL_Runtime_Bus.G_TX_Healthy
   AND GVL_Runtime_Bus.G_RX_Healthy THEN

    GVL_Cluster_Runtime_FSM.G_State_Synchronization := TRUE;

END_IF;

// Operational state.
IF GVL_Distributed_Execution_Gates.G_Can_Execute
   AND GVL_Distributed_Execution_Gates.G_Can_Orchestrate
   AND L_Finalized_Runtime_Continuity THEN

    GVL_Cluster_Runtime_FSM.G_State_Operational := TRUE;

    GVL_Cluster_Runtime_FSM.G_Status_Code := 0;
    GVL_Cluster_Runtime_FSM.G_Status_Text :=
        'Cluster runtime operational';

END_IF;

// Degraded state.
IF GVL_Cluster_Safety_Barrier.G_Cluster_Execution_Blocked THEN

    GVL_Cluster_Runtime_FSM.G_State_Degraded := TRUE;

    GVL_Cluster_Runtime_FSM.G_Status_Code := 10;
    GVL_Cluster_Runtime_FSM.G_Status_Text :=
        'Cluster runtime degraded';

END_IF;

// Observer-only state.
IF GVL_Distributed_Authority.G_Authority_State.Authority_Observer_Only THEN

    GVL_Cluster_Runtime_FSM.G_State_Observer_Only := TRUE;

    GVL_Cluster_Runtime_FSM.G_Status_Code := 11;
    GVL_Cluster_Runtime_FSM.G_Status_Text :=
        'Cluster runtime observer-only';

END_IF;

// Recovery lock state.
IF GVL_Distributed_Recovery_Lock.G_Recovery_Execution_Blocked THEN

    GVL_Cluster_Runtime_FSM.G_State_Recovery_Lock := TRUE;

    GVL_Cluster_Runtime_FSM.G_Status_Code := 12;
    GVL_Cluster_Runtime_FSM.G_Status_Text :=
        'Cluster runtime recovery-locked';

END_IF;

// Quarantine state.
IF GVL_Runtime_Discovery.G_Any_Node_Quarantined THEN

    GVL_Cluster_Runtime_FSM.G_State_Quarantine := TRUE;

    GVL_Cluster_Runtime_FSM.G_Status_Code := 13;
    GVL_Cluster_Runtime_FSM.G_Status_Text :=
        'Cluster runtime quarantined';

END_IF;

GVL_Cluster_Runtime_FSM.G_Runtime_Valid := TRUE;
GVL_Cluster_Runtime_FSM.G_Last_Update_MS := VI_System_Time_MS;

END_FUNCTION_BLOCK

(* ---- FB_Cluster_Safety_Barrier_Runtime.st ---- *)
FUNCTION_BLOCK FB_Cluster_Safety_Barrier_Runtime
VAR_INPUT
    VI_Enable : BOOL;
    VI_System_Time_MS : UDINT;
END_VAR
VAR
    L_Block_Execution : BOOL;
    L_Status_Code : UINT;
    L_Status_Text : STRING(160);

    L_Finalized_Runtime_Continuity : BOOL;
END_VAR

IF NOT VI_Enable THEN
    GVL_Cluster_Safety_Barrier.G_Runtime_Valid := FALSE;
    RETURN;
END_IF;

L_Block_Execution := FALSE;
L_Status_Code := 0;
L_Status_Text := 'Cluster safety barrier healthy';

GVL_Cluster_Safety_Barrier.G_Remote_Authority_Degraded := FALSE;
GVL_Cluster_Safety_Barrier.G_Runtime_Bus_Degraded := FALSE;
GVL_Cluster_Safety_Barrier.G_Projection_Ownership_Invalid := FALSE;
GVL_Cluster_Safety_Barrier.G_Recovery_Lock_Active := FALSE;
GVL_Cluster_Safety_Barrier.G_Deployment_Invalid := FALSE;
GVL_Cluster_Safety_Barrier.G_Authority_Downgraded := FALSE;
GVL_Cluster_Safety_Barrier.G_Orchestration_Restricted := FALSE;

// Finalized runtime continuity proof chain.
L_Finalized_Runtime_Continuity :=
    GVL_SEMANTIC_PROGRESS.Semantic_Forward_Progress_Valid
    AND GVL_SEMANTIC_PROGRESS.Semantic_Execution_Continuity_OK
    AND NOT GVL_SEMANTIC_PROGRESS.Semantic_Progress_Lease_Expired
    AND NOT GVL_SEMANTIC_PROGRESS.Semantic_Progress_Quarantine_Active
    AND GVL_RUNTIME_SNAPSHOT.Snapshot_Frozen
    AND GVL_RUNTIME_SNAPSHOT.Snapshot_Publication_Allowed
    AND GVL_RUNTIME_SNAPSHOT.Snapshot_Copy_Valid
    AND GVL_RUNTIME_SNAPSHOT.Snapshot_Isolation_Valid
    AND NOT GVL_RUNTIME_SNAPSHOT.Snapshot_Mutation_Detected
    AND GVL_DISTRIBUTED_SNAPSHOT.Distributed_Publication_Reconciled
    AND GVL_DISTRIBUTED_SNAPSHOT.Distributed_Publication_Freeze_Valid
    AND GVL_DISTRIBUTED_SNAPSHOT.Distributed_Snapshot_Consistent
    AND GVL_DISTRIBUTED_COMMIT.Distributed_Commit_Valid
    AND GVL_DISTRIBUTED_COMMIT.Publication_Prepare_Valid
    AND GVL_DISTRIBUTED_COMMIT.Publication_Commit_Confirmed
    AND NOT GVL_DISTRIBUTED_COMMIT.Peer_Commit_Mismatch
    AND NOT GVL_DISTRIBUTED_COMMIT.Commit_Lease_Expired
    AND GVL_OUTPUT_EPOCH.Output_Publication_Valid
    AND GVL_OUTPUT_EPOCH.Output_Runtime_Epoch_Valid
    AND NOT GVL_OUTPUT_EPOCH.Output_Lease_Expired
    AND NOT GVL_OUTPUT_EPOCH.Output_Forced_Safe_Decay
    AND GVL_COMMAND_VERIFY.PreOutput_Barrier_OK
    AND NOT GVL_COMMAND_VERIFY.PreOutput_Block_IO;

// Root finalized continuity barrier.
IF NOT L_Finalized_Runtime_Continuity THEN

    L_Block_Execution := TRUE;
    L_Status_Code := 9;
    L_Status_Text :=
        'Finalized runtime continuity invalid';

    GVL_Cluster_Safety_Barrier.G_Authority_Downgraded := TRUE;
    GVL_Cluster_Safety_Barrier.G_Orchestration_Restricted := TRUE;

END_IF;

// Remote authority staleness barrier.
IF GVL_Distributed_Runtime.G_Any_Remote_Node_Offline
   OR GVL_Distributed_Runtime.G_Split_Brain_Suspected THEN

    L_Block_Execution := TRUE;
    L_Status_Code := 10;
    L_Status_Text :=
        'Cluster authority state degraded';

    GVL_Cluster_Safety_Barrier.G_Remote_Authority_Degraded := TRUE;

END_IF;

// Runtime bus integrity barrier.
IF GVL_Runtime_Bus.G_Any_Replication_Rejected
   OR NOT GVL_Runtime_Bus.G_TX_Healthy
   OR NOT GVL_Runtime_Bus.G_RX_Healthy THEN

    L_Block_Execution := TRUE;
    L_Status_Code := 11;
    L_Status_Text :=
        'Runtime bus integrity degraded';

    GVL_Cluster_Safety_Barrier.G_Runtime_Bus_Degraded := TRUE;

END_IF;

// Projection ownership barrier.
IF GVL_Distributed_Projection_Ownership.G_Any_Ownership_Conflict
   OR GVL_Distributed_Projection_Ownership.G_Any_Ownership_Stale THEN

    L_Block_Execution := TRUE;
    L_Status_Code := 12;
    L_Status_Text :=
        'Distributed projection ownership invalid';

    GVL_Cluster_Safety_Barrier.G_Projection_Ownership_Invalid := TRUE;

END_IF;

// Recovery lock barrier.
IF GVL_Distributed_Recovery_Lock.G_Recovery_Execution_Blocked
   OR GVL_Distributed_Recovery_Lock.G_Rollback_Execution_Blocked
   OR GVL_Distributed_Recovery_Lock.G_Reopen_Execution_Blocked THEN

    L_Block_Execution := TRUE;
    L_Status_Code := 13;
    L_Status_Text :=
        'Distributed recovery execution blocked';

    GVL_Cluster_Safety_Barrier.G_Recovery_Lock_Active := TRUE;

END_IF;

// Discovery/deployment barrier.
IF GVL_Runtime_Discovery.G_Any_Discovery_Rejected
   OR GVL_Runtime_Discovery.G_Any_Node_Quarantined THEN

    L_Block_Execution := TRUE;
    L_Status_Code := 14;
    L_Status_Text :=
        'Runtime deployment/discovery invalid';

    GVL_Cluster_Safety_Barrier.G_Deployment_Invalid := TRUE;

END_IF;

// Cluster escalation semantics.
IF L_Block_Execution THEN

    GVL_Distributed_Authority.G_Authority_State.Authority_Observer_Only := TRUE;
    GVL_Distributed_Authority.G_Authority_State.Authority_Master_Elected := FALSE;

    GVL_Distributed_Orchestration.G_Distributed_Projection_Healthy := FALSE;

    GVL_Cluster_Safety_Barrier.G_Authority_Downgraded := TRUE;
    GVL_Cluster_Safety_Barrier.G_Orchestration_Restricted := TRUE;

END_IF;

GVL_Cluster_Safety_Barrier.G_Cluster_Execution_Blocked :=
    L_Block_Execution;

GVL_Cluster_Safety_Barrier.G_Runtime_Valid := TRUE;
GVL_Cluster_Safety_Barrier.G_Last_Update_MS := VI_System_Time_MS;
GVL_Cluster_Safety_Barrier.G_Status_Code := L_Status_Code;
GVL_Cluster_Safety_Barrier.G_Status_Text := L_Status_Text;

END_FUNCTION_BLOCK

(* ---- FB_Device_Predictive_Diag.st ---- *)
FUNCTION_BLOCK FB_Device_Predictive_Diag
VAR_INPUT
    VI_Current_Value : REAL;      // Текущий ток или время
    VI_Nominal_Value : REAL;      // Эталонное значение
    VI_Is_Running    : BOOL;
    VI_Reset_Stats   : BOOL;
    VI_System_Time_MS: UDINT;     // Системное время (мс)
END_VAR
VAR_IN_OUT
    VIO_Health_Data  : ST_Device_Health;
END_VAR
VAR
    L_Prev_Running   : BOOL;
    L_Start_Time     : UDINT;
    L_Last_Calc_Time : UDINT;
    L_Elapsed_MS     : UDINT;
    L_Accumulated_MS : UDINT; // Накопленное время работы (мс)
    L_Timer_Running  : FB_System_Timer;
END_VAR

// 0. Сброс статистики
IF VI_Reset_Stats THEN
    VIO_Health_Data.Starts_Count := 0;
    VIO_Health_Data.Sample_Count := 0;
    VIO_Health_Data.Current_Sum := 0.0;
    VIO_Health_Data.Avg_Start_Current := 0.0;
    VIO_Health_Data.Health_Score := 100;
    VIO_Health_Data.Maintenance_Required := FALSE;
    VIO_Health_Data.Warning_Message := '';
    VIO_Health_Data.Last_Start_Current := 0.0;
    VIO_Health_Data.Total_Runtime_Hours := 0;
    L_Accumulated_MS := 0;
END_IF;

// 1. Счётчик пусков и замер пускового тока
IF VI_Is_Running AND NOT L_Prev_Running THEN
    VIO_Health_Data.Starts_Count := VIO_Health_Data.Starts_Count + 1;
    VIO_Health_Data.Last_Start_Current := VI_Current_Value;
    L_Start_Time := VI_System_Time_MS;
    L_Last_Calc_Time := VI_System_Time_MS;

    // Обновление среднего пускового тока
    VIO_Health_Data.Sample_Count := VIO_Health_Data.Sample_Count + 1;
    VIO_Health_Data.Current_Sum := VIO_Health_Data.Current_Sum + VI_Current_Value;
    VIO_Health_Data.Avg_Start_Current := VIO_Health_Data.Current_Sum / UDINT_TO_REAL(VIO_Health_Data.Sample_Count);

    // 2. Анализ отклонения пускового тока (п. 12.1 ТЗ)
    IF VI_Current_Value > (VI_Nominal_Value * 1.5) THEN
        VIO_Health_Data.Health_Score := TO_BYTE(LIMIT(0, TO_INT(VIO_Health_Data.Health_Score) - 5, 100));
    ELSIF VI_Current_Value > (VI_Nominal_Value * 1.2) THEN
        VIO_Health_Data.Health_Score := TO_BYTE(LIMIT(0, TO_INT(VIO_Health_Data.Health_Score) - 1, 100));
    ELSIF VI_Current_Value < (VI_Nominal_Value * 0.5) THEN
        VIO_Health_Data.Health_Score := TO_BYTE(LIMIT(0, TO_INT(VIO_Health_Data.Health_Score) - 2, 100));
    END_IF;
END_IF;

// 3. Анализ рабочего тока и наработки
IF VI_Is_Running THEN
    L_Elapsed_MS := (VI_System_Time_MS - L_Last_Calc_Time);
    L_Accumulated_MS := L_Accumulated_MS + L_Elapsed_MS;
    L_Last_Calc_Time := VI_System_Time_MS;

    // Обновляем наработку каждый час (3600000 мс)
    IF L_Accumulated_MS >= 3600000 THEN
        VIO_Health_Data.Total_Runtime_Hours := VIO_Health_Data.Total_Runtime_Hours + 1;
        L_Accumulated_MS := L_Accumulated_MS - 3600000;

        // Естественный износ: -1% здоровья каждые 1000 часов
        IF (VIO_Health_Data.Total_Runtime_Hours MOD 1000) = 0 THEN
            VIO_Health_Data.Health_Score := TO_BYTE(LIMIT(0, TO_INT(VIO_Health_Data.Health_Score) - 1, 100));
        END_IF;

        // Анализ рабочего тока (после пускового режима)
        IF (VI_System_Time_MS - L_Start_Time) > 10000 THEN // 10 секунд после пуска
            IF VI_Current_Value > (VI_Nominal_Value * 1.1) THEN
                // Повышенный рабочий ток - ускоренный износ (-1% в час)
                VIO_Health_Data.Health_Score := TO_BYTE(LIMIT(0, TO_INT(VIO_Health_Data.Health_Score) - 1, 100));
            END_IF;
        END_IF;
    END_IF;
END_IF;

// 4. Генерация предупреждения
IF VIO_Health_Data.Health_Score < 20 THEN
    VIO_Health_Data.Maintenance_Required := TRUE;
    VIO_Health_Data.Warning_Message := 'Критический износ: проверьте механику';
ELSIF VIO_Health_Data.Health_Score < 60 THEN
    VIO_Health_Data.Maintenance_Required := FALSE;
    VIO_Health_Data.Warning_Message := 'Предупреждение: повышенное трение';
ELSE
    VIO_Health_Data.Maintenance_Required := FALSE;
    VIO_Health_Data.Warning_Message := 'В норме';
END_IF;

L_Prev_Running := VI_Is_Running;
END_FUNCTION_BLOCK

(* ---- FB_Distributed_Execution_Gates_Runtime.st ---- *)
FUNCTION_BLOCK FB_Distributed_Execution_Gates_Runtime
VAR_INPUT
    VI_Enable : BOOL;
    VI_System_Time_MS : UDINT;
END_VAR
VAR
    L_Allow : BOOL;
    L_Observer_Only : BOOL;

    L_Semantic_Continuity_Valid : BOOL;
    L_Finalized_Publication_Continuity : BOOL;
END_VAR

IF NOT VI_Enable THEN
    GVL_Distributed_Execution_Gates.G_Runtime_Valid := FALSE;
    RETURN;
END_IF;

// Observer-only runtime semantics.
// Observer nodes may:
//   - observe runtime state;
//   - receive publications;
//   - participate in diagnostics.
//
// Observer nodes must NEVER:
//   - execute orchestration;
//   - own projections;
//   - execute recovery;
//   - publish physical outputs.
L_Observer_Only :=
    GVL_Distributed_Authority.G_Authority_State.Authority_Observer_Only;

// Semantic continuity authority.
L_Semantic_Continuity_Valid :=
    GVL_SEMANTIC_PROGRESS.Semantic_Forward_Progress_Valid
    AND GVL_SEMANTIC_PROGRESS.Semantic_Execution_Continuity_OK
    AND NOT GVL_SEMANTIC_PROGRESS.Semantic_Progress_Lease_Expired
    AND NOT GVL_SEMANTIC_PROGRESS.Semantic_Progress_Quarantine_Active
    AND NOT GVL_SEMANTIC_PROGRESS.Semantic_Replay_Suspected
    AND NOT GVL_SEMANTIC_PROGRESS.Semantic_Livelock_Suspected
    AND NOT GVL_SEMANTIC_PROGRESS.Semantic_Deadlock_Suspected;

// Finalized publication proof chain.
L_Finalized_Publication_Continuity :=
    GVL_RUNTIME_SNAPSHOT.Snapshot_Frozen
    AND GVL_RUNTIME_SNAPSHOT.Snapshot_Publication_Allowed
    AND GVL_RUNTIME_SNAPSHOT.Snapshot_Copy_Valid
    AND GVL_RUNTIME_SNAPSHOT.Snapshot_Isolation_Valid
    AND NOT GVL_RUNTIME_SNAPSHOT.Snapshot_Mutation_Detected
    AND GVL_DISTRIBUTED_SNAPSHOT.Distributed_Publication_Reconciled
    AND GVL_DISTRIBUTED_SNAPSHOT.Distributed_Publication_Freeze_Valid
    AND GVL_DISTRIBUTED_SNAPSHOT.Distributed_Snapshot_Consistent
    AND GVL_DISTRIBUTED_COMMIT.Distributed_Commit_Valid
    AND GVL_DISTRIBUTED_COMMIT.Publication_Prepare_Valid
    AND GVL_DISTRIBUTED_COMMIT.Publication_Commit_Confirmed
    AND NOT GVL_DISTRIBUTED_COMMIT.Peer_Commit_Mismatch
    AND NOT GVL_DISTRIBUTED_COMMIT.Commit_Lease_Expired
    AND GVL_OUTPUT_EPOCH.Output_Publication_Valid
    AND GVL_OUTPUT_EPOCH.Output_Runtime_Epoch_Valid
    AND NOT GVL_OUTPUT_EPOCH.Output_Lease_Expired
    AND NOT GVL_OUTPUT_EPOCH.Output_Forced_Safe_Decay
    AND GVL_COMMAND_VERIFY.PreOutput_Barrier_OK
    AND NOT GVL_COMMAND_VERIFY.PreOutput_Block_IO;

L_Allow :=
    NOT GVL_Cluster_Safety_Barrier.G_Cluster_Execution_Blocked
    AND GVL_Distributed_Authority.G_Authority_State.Authority_Master_Elected
    AND NOT GVL_Distributed_Runtime.G_Split_Brain_Suspected
    AND NOT GVL_Distributed_Projection_Ownership.G_Any_Ownership_Conflict
    AND NOT GVL_Runtime_Sessions.G_Any_Stale_Session
    AND L_Semantic_Continuity_Valid
    AND L_Finalized_Publication_Continuity
    AND NOT L_Observer_Only;

GVL_Distributed_Execution_Gates.G_Can_Replicate :=
    GVL_Runtime_Bus.G_TX_Healthy
    AND GVL_Runtime_Bus.G_RX_Healthy;

GVL_Distributed_Execution_Gates.G_Can_Execute :=
    L_Allow;

GVL_Distributed_Execution_Gates.G_Can_Orchestrate :=
    L_Allow
    AND GVL_Distributed_Orchestration.G_Distributed_Scheduler_Healthy;

GVL_Distributed_Execution_Gates.G_Can_Recover :=
    L_Allow
    AND NOT GVL_Distributed_Recovery_Lock.G_Recovery_Execution_Blocked;

GVL_Distributed_Execution_Gates.G_Can_Rollback :=
    L_Allow
    AND NOT GVL_Distributed_Recovery_Lock.G_Rollback_Execution_Blocked;

GVL_Distributed_Execution_Gates.G_Can_Own_Projection :=
    L_Allow
    AND NOT GVL_Distributed_Projection_Ownership.G_Any_Projection_Blocked;

GVL_Distributed_Execution_Gates.G_Runtime_Valid := TRUE;
GVL_Distributed_Execution_Gates.G_Last_Update_MS :=
    VI_System_Time_MS;

IF L_Observer_Only THEN

    GVL_Distributed_Execution_Gates.G_Status_Code := 2;
    GVL_Distributed_Execution_Gates.G_Status_Text :=
        'Distributed runtime observer-only';

ELSIF L_Allow THEN

    GVL_Distributed_Execution_Gates.G_Status_Code := 0;
    GVL_Distributed_Execution_Gates.G_Status_Text :=
        'Distributed execution gates open';

ELSE

    GVL_Distributed_Execution_Gates.G_Status_Code := 1;
    GVL_Distributed_Execution_Gates.G_Status_Text :=
        'Distributed execution gates restricted';

END_IF;

END_FUNCTION_BLOCK

(* ---- FB_Distributed_Orchestration_Runtime.st ---- *)
FUNCTION_BLOCK FB_Distributed_Orchestration_Runtime
VAR_INPUT
    VI_Enable : BOOL;
    VI_System_Time_MS : UDINT;
END_VAR
VAR
    L_State : ST_Distributed_Orchestration_State;
    L_Finalized_Runtime_Continuity : BOOL;
END_VAR

IF NOT VI_Enable THEN
    GVL_Distributed_Orchestration.G_Runtime_Valid := FALSE;
    RETURN;
END_IF;

L_State.Runtime_Valid := TRUE;
L_State.Runtime_System_Time_MS := VI_System_Time_MS;

L_State.Orchestration_Sequence_Id :=
    GVL_Distributed_Orchestration.G_Last_Distributed_Sequence_Id + 1;

L_State.Distributed_Execution_Active := TRUE;

L_State.Cross_Node_Isolation_Required :=
    GVL_Distributed_Orchestration.G_Cross_Node_Isolation_Active;

L_State.Cross_Node_Recovery_Required :=
    GVL_Distributed_Orchestration.G_Cross_Node_Recovery_Active;

L_State.Cross_Node_Rollback_Required :=
    GVL_Distributed_Orchestration.G_Cross_Node_Rollback_Active;

L_Finalized_Runtime_Continuity :=
    GVL_SEMANTIC_PROGRESS.Semantic_Forward_Progress_Valid
    AND GVL_SEMANTIC_PROGRESS.Semantic_Execution_Continuity_OK
    AND NOT GVL_SEMANTIC_PROGRESS.Semantic_Progress_Lease_Expired
    AND NOT GVL_SEMANTIC_PROGRESS.Semantic_Progress_Quarantine_Active
    AND GVL_RUNTIME_SNAPSHOT.Snapshot_Frozen
    AND GVL_RUNTIME_SNAPSHOT.Snapshot_Publication_Allowed
    AND GVL_RUNTIME_SNAPSHOT.Snapshot_Copy_Valid
    AND GVL_RUNTIME_SNAPSHOT.Snapshot_Isolation_Valid
    AND NOT GVL_RUNTIME_SNAPSHOT.Snapshot_Mutation_Detected
    AND GVL_DISTRIBUTED_SNAPSHOT.Distributed_Publication_Reconciled
    AND GVL_DISTRIBUTED_SNAPSHOT.Distributed_Publication_Freeze_Valid
    AND GVL_DISTRIBUTED_SNAPSHOT.Distributed_Snapshot_Consistent
    AND GVL_DISTRIBUTED_COMMIT.Distributed_Commit_Valid
    AND GVL_DISTRIBUTED_COMMIT.Publication_Prepare_Valid
    AND GVL_DISTRIBUTED_COMMIT.Publication_Commit_Confirmed
    AND NOT GVL_DISTRIBUTED_COMMIT.Peer_Commit_Mismatch
    AND NOT GVL_DISTRIBUTED_COMMIT.Commit_Lease_Expired
    AND GVL_OUTPUT_EPOCH.Output_Publication_Valid
    AND GVL_OUTPUT_EPOCH.Output_Runtime_Epoch_Valid
    AND NOT GVL_OUTPUT_EPOCH.Output_Lease_Expired
    AND NOT GVL_OUTPUT_EPOCH.Output_Forced_Safe_Decay
    AND GVL_COMMAND_VERIFY.PreOutput_Barrier_OK
    AND NOT GVL_COMMAND_VERIFY.PreOutput_Block_IO;

L_State.Distributed_Scheduler_Healthy :=
    GVL_Runtime_Bus.G_TX_Healthy
    AND GVL_Distributed_Runtime.G_Distributed_Authority_Healthy
    AND L_Finalized_Runtime_Continuity;

L_State.Distributed_Timing_Window_Valid :=
    GVL_Distributed_Authority.G_Distributed_Safety_Barrier_OK
    AND L_Finalized_Runtime_Continuity;

IF L_State.Distributed_Scheduler_Healthy
   AND L_State.Distributed_Timing_Window_Valid THEN
    L_State.Distributed_Projection_Granted := TRUE;
    L_State.Distributed_Recovery_Allowed := TRUE;
    L_State.Distributed_Rollback_Allowed := TRUE;
    L_State.Status_Code := 0;
    L_State.Status_Text := 'Distributed orchestration runtime healthy';
ELSE
    L_State.Distributed_Projection_Blocked := TRUE;
    L_State.Distributed_Conflict_Detected := TRUE;
    L_State.Status_Code := 2;
    L_State.Status_Text := 'Distributed orchestration blocked';
END_IF;

IF GVL_Distributed_Runtime.G_Split_Brain_Suspected THEN
    L_State.Distributed_Split_Execution_Suspected := TRUE;
    L_State.Distributed_Projection_Blocked := TRUE;
    L_State.Status_Code := 3;
    L_State.Status_Text := 'Distributed split execution suspected';
END_IF;

GVL_Distributed_Orchestration.G_Orchestration_State := L_State;
GVL_Distributed_Orchestration.G_Last_Distributed_Sequence_Id := L_State.Orchestration_Sequence_Id;
GVL_Distributed_Orchestration.G_Distributed_Projection_Healthy := L_State.Distributed_Projection_Granted;
GVL_Distributed_Orchestration.G_Distributed_Scheduler_Healthy := L_State.Distributed_Scheduler_Healthy;
GVL_Distributed_Orchestration.G_Runtime_Valid := TRUE;
GVL_Distributed_Orchestration.G_Last_Update_MS := VI_System_Time_MS;
GVL_Distributed_Orchestration.G_Status_Code := L_State.Status_Code;
GVL_Distributed_Orchestration.G_Status_Text := L_State.Status_Text;

END_FUNCTION_BLOCK

(* ---- FB_Distributed_Runtime_Continuity.st ---- *)
FUNCTION_BLOCK FB_Distributed_Runtime_Continuity
VAR_INPUT
    VI_Enable : BOOL;
    VI_System_Time_MS : UDINT;
END_VAR
VAR
    L_i : INT;
    L_Node : ST_Distributed_Runtime_Node_State;

    L_Any_Offline : BOOL;
    L_Any_Degraded : BOOL;
    L_Split_Brain : BOOL;

    L_Finalized_Runtime_Continuity : BOOL;
END_VAR

IF NOT VI_Enable THEN
    GVL_Distributed_Runtime.G_Runtime_Valid := FALSE;
    RETURN;
END_IF;

// Finalized runtime continuity proof chain.
L_Finalized_Runtime_Continuity :=
    GVL_SEMANTIC_PROGRESS.Semantic_Forward_Progress_Valid
    AND GVL_SEMANTIC_PROGRESS.Semantic_Execution_Continuity_OK
    AND NOT GVL_SEMANTIC_PROGRESS.Semantic_Progress_Lease_Expired
    AND NOT GVL_SEMANTIC_PROGRESS.Semantic_Progress_Quarantine_Active
    AND GVL_RUNTIME_SNAPSHOT.Snapshot_Frozen
    AND GVL_RUNTIME_SNAPSHOT.Snapshot_Publication_Allowed
    AND GVL_RUNTIME_SNAPSHOT.Snapshot_Copy_Valid
    AND GVL_RUNTIME_SNAPSHOT.Snapshot_Isolation_Valid
    AND NOT GVL_RUNTIME_SNAPSHOT.Snapshot_Mutation_Detected
    AND GVL_DISTRIBUTED_SNAPSHOT.Distributed_Publication_Reconciled
    AND GVL_DISTRIBUTED_SNAPSHOT.Distributed_Publication_Freeze_Valid
    AND GVL_DISTRIBUTED_SNAPSHOT.Distributed_Snapshot_Consistent
    AND GVL_DISTRIBUTED_COMMIT.Distributed_Commit_Valid
    AND GVL_DISTRIBUTED_COMMIT.Publication_Prepare_Valid
    AND GVL_DISTRIBUTED_COMMIT.Publication_Commit_Confirmed
    AND NOT GVL_DISTRIBUTED_COMMIT.Peer_Commit_Mismatch
    AND NOT GVL_DISTRIBUTED_COMMIT.Commit_Lease_Expired
    AND GVL_OUTPUT_EPOCH.Output_Publication_Valid
    AND GVL_OUTPUT_EPOCH.Output_Runtime_Epoch_Valid
    AND NOT GVL_OUTPUT_EPOCH.Output_Lease_Expired
    AND NOT GVL_OUTPUT_EPOCH.Output_Forced_Safe_Decay
    AND GVL_COMMAND_VERIFY.PreOutput_Barrier_OK
    AND NOT GVL_COMMAND_VERIFY.PreOutput_Block_IO;

// Local node authoritative runtime state.
GVL_Distributed_Runtime.G_Local_Node_State.Runtime_Valid := TRUE;
GVL_Distributed_Runtime.G_Local_Node_State.Runtime_System_Time_MS :=
    VI_System_Time_MS;

GVL_Distributed_Runtime.G_Local_Node_State.Node_Online :=
    L_Finalized_Runtime_Continuity;

GVL_Distributed_Runtime.G_Local_Node_State.Restart_Continuity_Valid :=
    GVL_Runtime_Restart_Continuity.G_Runtime_Valid
    AND L_Finalized_Runtime_Continuity;

GVL_Distributed_Runtime.G_Local_Node_State.Quarantine_State_Replicated :=
    NOT GVL_Config_Activation.G_Config_Quarantine_Active
    AND L_Finalized_Runtime_Continuity;

GVL_Distributed_Runtime.G_Local_Node_State.Recovery_State_Replicated :=
    GVL_Water_Recovery_Runtime.G_Runtime_Valid
    AND L_Finalized_Runtime_Continuity;

GVL_Distributed_Runtime.G_Local_Node_State.Authority_Allowed :=
    NOT GVL_COMMAND_VERIFY.PreOutput_Block_IO
    AND L_Finalized_Runtime_Continuity;

GVL_Distributed_Runtime.G_Local_Node_State.Replication_Healthy :=
    L_Finalized_Runtime_Continuity;

FOR L_i := 1 TO 8 DO

    L_Node := GVL_Distributed_Runtime.G_Remote_Node_State[L_i];

    IF L_Node.Runtime_Valid THEN

        IF NOT L_Node.Node_Online THEN
            L_Any_Offline := TRUE;
        END_IF;

        IF L_Node.Node_Degraded
           OR L_Node.Node_Quarantined THEN

            L_Any_Degraded := TRUE;

        END_IF;

        IF L_Node.Authority_Master
           AND GVL_Distributed_Runtime.G_Local_Node_State.Authority_Master THEN

            L_Split_Brain := TRUE;

        END_IF;

    END_IF;

END_FOR;

IF NOT L_Finalized_Runtime_Continuity THEN
    L_Any_Degraded := TRUE;
END_IF;

GVL_Distributed_Runtime.G_Any_Remote_Node_Offline :=
    L_Any_Offline;

GVL_Distributed_Runtime.G_Any_Remote_Node_Degraded :=
    L_Any_Degraded;

GVL_Distributed_Runtime.G_Split_Brain_Suspected :=
    L_Split_Brain;

GVL_Distributed_Runtime.G_Distributed_Replication_Healthy :=
    NOT L_Any_Offline
    AND L_Finalized_Runtime_Continuity;

GVL_Distributed_Runtime.G_Distributed_Authority_Healthy :=
    NOT L_Split_Brain
    AND L_Finalized_Runtime_Continuity;

GVL_Distributed_Runtime.G_Runtime_Valid := TRUE;
GVL_Distributed_Runtime.G_Last_Update_MS := VI_System_Time_MS;

IF NOT L_Finalized_Runtime_Continuity THEN
    GVL_Distributed_Runtime.G_Status_Code := 4;
    GVL_Distributed_Runtime.G_Status_Text :=
        'Distributed finalized continuity invalid';
ELSIF L_Split_Brain THEN
    GVL_Distributed_Runtime.G_Status_Code := 3;
    GVL_Distributed_Runtime.G_Status_Text :=
        'Distributed split-brain suspected';
ELSIF L_Any_Degraded THEN
    GVL_Distributed_Runtime.G_Status_Code := 2;
    GVL_Distributed_Runtime.G_Status_Text :=
        'Distributed degraded node detected';
ELSIF L_Any_Offline THEN
    GVL_Distributed_Runtime.G_Status_Code := 1;
    GVL_Distributed_Runtime.G_Status_Text :=
        'Distributed offline node detected';
ELSE
    GVL_Distributed_Runtime.G_Status_Code := 0;
    GVL_Distributed_Runtime.G_Status_Text :=
        'Distributed runtime continuity healthy';
END_IF;

END_FUNCTION_BLOCK

(* ---- FB_Gas_Smoke_Manager.st ---- *)
FUNCTION_BLOCK FB_Gas_Smoke_Manager
VAR_INPUT
    VI_System_Time_MS : UDINT;
    VI_IsActivePLC    : BOOL;
    VI_Mute_Request   : BOOL;
END_VAR

VAR_IN_OUT
    VI_Methane_LEL    : ARRAY[1..GVL_CONSTANTS.C_MAX_METHANE_SENSORS] OF REAL;
    VI_CO_PPM         : ARRAY[1..GVL_CONSTANTS.C_MAX_CO_SENSORS] OF REAL;
    VI_Smoke_Sensors  : ARRAY[1..GVL_CONSTANTS.C_MAX_SMOKE_SENSORS] OF BOOL;
END_VAR

VAR_OUTPUT
    // Health signals
    VO_Smoke_Detected   : BOOL;
    VO_Gas_Detected     : BOOL;
    VO_CO_Warning_Level : BOOL;
    VO_CO_Alarm_Level   : BOOL;
    VO_Status_Msg       : STRING(200);
END_VAR

VAR
    L_Methane_Max   : REAL;
    L_CO_Max        : REAL;
    L_Smoke_Count   : UINT;
    L_Smoke_Active  : BOOL;
    L_i             : INT;

    L_CO_Timer_30ppm  : FB_System_Timer;
    L_CO_Timer_70ppm  : FB_System_Timer;
    L_CO_Timer_400ppm : FB_System_Timer;

    L_CO_Level_30   : BOOL;
    L_CO_Level_70   : BOOL;
    L_CO_Level_400  : BOOL;

    L_Smoke_Timer : ARRAY[1..GVL_CONSTANTS.C_MAX_SMOKE_SENSORS] OF FB_System_Timer;
END_VAR

IF NOT VI_IsActivePLC THEN RETURN; END_IF;

// Reset outputs
VO_Smoke_Detected := FALSE;
VO_Gas_Detected := FALSE;
VO_CO_Warning_Level := FALSE;
VO_CO_Alarm_Level := FALSE;
VO_Status_Msg := 'ОК';

// --- Methane ---
L_Methane_Max := 0.0;
FOR L_i := 1 TO GVL_CONSTANTS.C_MAX_METHANE_SENSORS DO
    IF VI_Methane_LEL[L_i] > L_Methane_Max THEN
        L_Methane_Max := VI_Methane_LEL[L_i];
    END_IF;
END_FOR;

IF L_Methane_Max >= 20.0 THEN
    VO_Gas_Detected := TRUE;
END_IF;

// --- CO ---
L_CO_Max := 0.0;
FOR L_i := 1 TO GVL_CONSTANTS.C_MAX_CO_SENSORS DO
    IF VI_CO_PPM[L_i] > L_CO_Max THEN
        L_CO_Max := VI_CO_PPM[L_i];
    END_IF;
END_FOR;

L_CO_Level_30 := (L_CO_Max >= 30.0);
L_CO_Level_70 := (L_CO_Max >= 70.0);
L_CO_Level_400 := (L_CO_Max >= 400.0);

L_CO_Timer_30ppm(IN := L_CO_Level_30, PT := T#8h, VI_System_Time_MS := VI_System_Time_MS);
L_CO_Timer_70ppm(IN := L_CO_Level_70, PT := T#1h, VI_System_Time_MS := VI_System_Time_MS);
L_CO_Timer_400ppm(IN := L_CO_Level_400, PT := T#15m, VI_System_Time_MS := VI_System_Time_MS);

IF L_CO_Timer_30ppm.Q THEN
    VO_CO_Warning_Level := TRUE;
END_IF;

IF L_CO_Timer_70ppm.Q OR L_CO_Timer_400ppm.Q THEN
    VO_CO_Alarm_Level := TRUE;
END_IF;

// --- Smoke ---
L_Smoke_Count := 0;
L_Smoke_Active := FALSE;

FOR L_i := 1 TO GVL_CONSTANTS.C_MAX_SMOKE_SENSORS DO
    L_Smoke_Timer[L_i](IN := VI_Smoke_Sensors[L_i], PT := T#30s, VI_System_Time_MS := VI_System_Time_MS);

    IF VI_Smoke_Sensors[L_i] THEN
        L_Smoke_Count := L_Smoke_Count + 1;
    END_IF;

    IF L_Smoke_Timer[L_i].Q OR (L_Smoke_Count >= 2) THEN
        L_Smoke_Active := TRUE;
    END_IF;
END_FOR;

IF L_Smoke_Active THEN
    VO_Smoke_Detected := TRUE;
END_IF;

// Status
IF VO_Smoke_Detected THEN
    VO_Status_Msg := 'ПОЖАР';
ELSIF VO_Gas_Detected THEN
    VO_Status_Msg := 'УТЕЧКА ГАЗА';
ELSIF VO_CO_Alarm_Level THEN
    VO_Status_Msg := 'КРИТИЧЕСКИЙ CO';
ELSIF VO_CO_Warning_Level THEN
    VO_Status_Msg := 'ПОВЫШЕННЫЙ CO';
ELSE
    VO_Status_Msg := 'ОК';
END_IF;
// >>> BULK_SYNC_ANCHOR: FB_Gas_Smoke_Manager <<<
END_FUNCTION_BLOCK

(* ---- FB_Heating_Circuit_Control.st ---- *)
// ==============================================================================
// Heating circuit control helper
//
// Internal refactoring helper for FB_Heating_System_Manager.
// Owns per-circuit sensor validation, temperature source fallback,
// floor-heating controller call, overheat shutdown, and rule action projection.
//
// Temperature source selection is confidence-aware:
// - range invalid still blocks that source;
// - passive input-quality confidence can prefer a healthier fallback;
// - degraded-but-range-valid sources remain operational if no better source exists.
//
// Publishes only canonical runtime projection semantics to
// GVL_Heating_Runtime_Projection. Explainability, predictive observation and
// supervisory ingestion consume that projection downstream.
// ==============================================================================
FUNCTION_BLOCK FB_Heating_Circuit_Control
VAR_INPUT
    VI_System_Time_MS : UDINT;
    VI_Current_Hour : UINT;
    VI_IsActivePLC : BOOL;
    VI_Config : ST_Heating_Config;
    VI_Tariff : ST_Tariff_Config;
    VI_Scenario_Adjust : REAL;
END_VAR

VAR_IN_OUT
    VI_Zone_Configs : ARRAY[1..GVL_CONSTANTS.C_MAX_HEATING_CIRCUITS] OF ST_FloorHeating_Circuit_Config;
    VI_Floor_Temps : ARRAY[1..GVL_CONSTANTS.C_MAX_HEATING_CIRCUITS] OF REAL;
    VI_Room_Temps : ARRAY[1..16] OF REAL;
    VI_Rule_Actions : ARRAY[1..GVL_CONSTANTS.C_MAX_RULES] OF ST_Rule_Action;
END_VAR

VAR_OUTPUT
    VO_Zone_Valves : ARRAY[1..GVL_CONSTANTS.C_MAX_HEATING_CIRCUITS] OF BOOL;
    VO_Heating_Sensor_Fault : BOOL;
END_VAR

VAR
    L_i : INT;
    L_j : INT;
    L_Climate_Zone_ID : INT;
    L_Zone_Config : ST_FloorHeating_Circuit_Config;
    L_Current_Temp : REAL;
    L_Sensor_Error : BOOL;
    L_Floor_Source_Valid : BOOL;
    L_Room_Source_Valid : BOOL;
    L_Floor_Confidence : REAL;
    L_Room_Confidence : REAL;
    L_Min_Source_Confidence : REAL;
    L_Primary_Source_Code : UINT;
    L_Selected_Source_Code : UINT;
    L_Primary_Confidence : REAL;
    L_Fallback_Confidence : REAL;
    L_Selected_Confidence : REAL;
    L_Fallback_Active : BOOL;
    L_Source_Degraded : BOOL;
    L_Reason_Code : UINT;
    L_Reason_Text : STRING(128);
    L_Selected_Source_Text : STRING(64);

    L_Prev_Selected_Source_Code : ARRAY[1..GVL_CONSTANTS.C_MAX_HEATING_CIRCUITS] OF UINT;
    L_Prev_Fallback_Active : ARRAY[1..GVL_CONSTANTS.C_MAX_HEATING_CIRCUITS] OF BOOL;
    L_Prev_Source_Loss : ARRAY[1..GVL_CONSTANTS.C_MAX_HEATING_CIRCUITS] OF BOOL;
    L_Source_Loss_Active : BOOL;

    L_Source_Switched_Event : BOOL;
    L_Fallback_Activated_Event : BOOL;
    L_Fallback_Recovered_Event : BOOL;
    L_Source_Loss_Event : BOOL;
    L_Last_Event_Code : UINT;
    L_Last_Event_Text : STRING(128);

    L_Floor_Controllers : ARRAY[1..GVL_CONSTANTS.C_MAX_HEATING_CIRCUITS] OF FB_FloorHeating_Controller;
    L_Overheat_Timer : ARRAY[1..GVL_CONSTANTS.C_MAX_HEATING_CIRCUITS] OF FB_System_Timer;
    fbFloorTempValidator : ARRAY[1..GVL_CONSTANTS.C_MAX_HEATING_CIRCUITS] OF FB_Analog_Validator;
    fbRoomTempValidator : ARRAY[1..16] OF FB_Analog_Validator;
END_VAR

VO_Heating_Sensor_Fault := FALSE;
L_Min_Source_Confidence := GVL_INPUT_VALIDATION_CONFIG.G_Min_Sensor_Confidence;

FOR L_i := 1 TO GVL_CONSTANTS.C_MAX_HEATING_CIRCUITS DO
    fbFloorTempValidator[L_i](
        VI_Value := VI_Floor_Temps[L_i],
        VI_Min_Valid := -40.0,
        VI_Max_Valid := 120.0,
        VI_Fallback_Mode := 0
    );

    L_Climate_Zone_ID := VI_Zone_Configs[L_i].zone;
    IF L_Climate_Zone_ID >= 1 AND L_Climate_Zone_ID <= 16 THEN
        fbRoomTempValidator[L_Climate_Zone_ID](
            VI_Value := VI_Room_Temps[L_Climate_Zone_ID],
            VI_Min_Valid := -40.0,
            VI_Max_Valid := 120.0,
            VI_Fallback_Mode := 0
        );
    END_IF;

    L_Floor_Source_Valid := NOT fbFloorTempValidator[L_i].VO_Error;
    L_Room_Source_Valid :=
        (L_Climate_Zone_ID >= 1) AND
        (L_Climate_Zone_ID <= 16) AND
        (NOT fbRoomTempValidator[L_Climate_Zone_ID].VO_Error);

    L_Floor_Confidence := REAL#1.0;
    IF GVL_INPUT_QUALITY.G_Floor_Temp_Quality[L_i].Quality_Visible THEN
        L_Floor_Confidence := GVL_INPUT_QUALITY.G_Floor_Temp_Quality[L_i].Confidence;
    END_IF;

    L_Room_Confidence := REAL#1.0;
    IF (L_Climate_Zone_ID >= 1) AND (L_Climate_Zone_ID <= 16) THEN
        IF GVL_INPUT_QUALITY.G_Room_Temp_Quality[L_Climate_Zone_ID].Quality_Visible THEN
            L_Room_Confidence := GVL_INPUT_QUALITY.G_Room_Temp_Quality[L_Climate_Zone_ID].Confidence;
        END_IF;
    END_IF;

    IF L_Floor_Confidence < REAL#0.0 THEN
        L_Floor_Confidence := REAL#0.0;
    ELSIF L_Floor_Confidence > REAL#1.0 THEN
        L_Floor_Confidence := REAL#1.0;
    END_IF;

    IF L_Room_Confidence < REAL#0.0 THEN
        L_Room_Confidence := REAL#0.0;
    ELSIF L_Room_Confidence > REAL#1.0 THEN
        L_Room_Confidence := REAL#1.0;
    END_IF;

    // Floor overheat protection remains floor-bound and range-validity based.
    L_Overheat_Timer[L_i](
        IN := L_Floor_Source_Valid AND (fbFloorTempValidator[L_i].VO_Value > VI_Config.Overheat_Threshold),
        PT := T#60s,
        VI_System_Time_MS := VI_System_Time_MS
    );

    L_Current_Temp := REAL#0.0;
    L_Sensor_Error := FALSE;
    L_Selected_Source_Code := 0;
    L_Selected_Source_Text := 'none';
    L_Selected_Confidence := REAL#0.0;
    L_Fallback_Active := FALSE;
    L_Source_Degraded := FALSE;
    L_Reason_Code := 0;
    L_Reason_Text := 'OK';

    IF VI_Zone_Configs[L_i].control_type = 1 OR VI_Zone_Configs[L_i].control_type = 2 THEN
        L_Primary_Source_Code := 1; // room
        L_Primary_Confidence := L_Room_Confidence;
        L_Fallback_Confidence := L_Floor_Confidence;

        // Primary: room air temperature. If room quality is degraded and floor
        // source is healthier, prefer floor fallback without declaring hard fault.
        IF L_Room_Source_Valid AND
           ((L_Room_Confidence >= L_Min_Source_Confidence) OR NOT L_Floor_Source_Valid OR (L_Room_Confidence >= L_Floor_Confidence)) THEN
            L_Current_Temp := fbRoomTempValidator[L_Climate_Zone_ID].VO_Value;
            L_Selected_Source_Code := 1;
            L_Selected_Source_Text := 'room';
            L_Selected_Confidence := L_Room_Confidence;
        ELSIF L_Floor_Source_Valid THEN
            L_Current_Temp := fbFloorTempValidator[L_i].VO_Value;
            L_Selected_Source_Code := 2;
            L_Selected_Source_Text := 'floor';
            L_Selected_Confidence := L_Floor_Confidence;
            L_Fallback_Active := TRUE;
        ELSIF L_Room_Source_Valid THEN
            L_Current_Temp := fbRoomTempValidator[L_Climate_Zone_ID].VO_Value;
            L_Selected_Source_Code := 1;
            L_Selected_Source_Text := 'room';
            L_Selected_Confidence := L_Room_Confidence;
            L_Source_Degraded := TRUE;
            L_Reason_Code := 2;
            L_Reason_Text := 'Room source degraded but retained; floor source unavailable';
        ELSE
            L_Sensor_Error := TRUE;
        END_IF;
    ELSE
        L_Primary_Source_Code := 2; // floor
        L_Primary_Confidence := L_Floor_Confidence;
        L_Fallback_Confidence := L_Room_Confidence;

        // Primary: floor temperature. If floor quality is degraded and room
        // source is healthier, prefer room fallback without declaring hard fault.
        IF L_Floor_Source_Valid AND
           ((L_Floor_Confidence >= L_Min_Source_Confidence) OR NOT L_Room_Source_Valid OR (L_Floor_Confidence >= L_Room_Confidence)) THEN
            L_Current_Temp := fbFloorTempValidator[L_i].VO_Value;
            L_Selected_Source_Code := 2;
            L_Selected_Source_Text := 'floor';
            L_Selected_Confidence := L_Floor_Confidence;
        ELSIF L_Room_Source_Valid THEN
            L_Current_Temp := fbRoomTempValidator[L_Climate_Zone_ID].VO_Value;
            L_Selected_Source_Code := 1;
            L_Selected_Source_Text := 'room';
            L_Selected_Confidence := L_Room_Confidence;
            L_Fallback_Active := TRUE;
        ELSIF L_Floor_Source_Valid THEN
            L_Current_Temp := fbFloorTempValidator[L_i].VO_Value;
            L_Selected_Source_Code := 2;
            L_Selected_Source_Text := 'floor';
            L_Selected_Confidence := L_Floor_Confidence;
            L_Source_Degraded := TRUE;
            L_Reason_Code := 2;
            L_Reason_Text := 'Floor source degraded but retained; room source unavailable';
        ELSE
            L_Sensor_Error := TRUE;
        END_IF;
    END_IF;

    IF L_Fallback_Active THEN
        L_Source_Degraded := TRUE;
        L_Reason_Code := 1;
        IF L_Primary_Source_Code = 1 THEN
            L_Reason_Text := 'Room source degraded or unavailable; floor fallback selected';
        ELSE
            L_Reason_Text := 'Floor source degraded or unavailable; room fallback selected';
        END_IF;
    END_IF;

    IF L_Sensor_Error THEN
        L_Source_Degraded := TRUE;
        L_Reason_Code := 3;
        L_Reason_Text := 'No valid temperature source available';
        VO_Heating_Sensor_Fault := TRUE;
        VO_Zone_Valves[L_i] := FALSE;
    ELSE
        L_Zone_Config := VI_Zone_Configs[L_i];
        L_Zone_Config.design_temp := L_Zone_Config.design_temp + VI_Scenario_Adjust;

        L_Floor_Controllers[L_i](
            VI_Current_Temp := L_Current_Temp,
            VI_Config := L_Zone_Config,
            VI_Tariff := VI_Tariff,
            VI_Current_Hour := VI_Current_Hour,
            VI_IsActivePLC := VI_IsActivePLC,
            VI_System_Time_MS := VI_System_Time_MS,
            VO_Valve_Bool => VO_Zone_Valves[L_i]
        );
    END_IF;

    L_Source_Loss_Active := L_Sensor_Error;

    L_Source_Switched_Event :=
        (L_Prev_Selected_Source_Code[L_i] <> 0) AND
        (L_Selected_Source_Code <> 0) AND
        (L_Selected_Source_Code <> L_Prev_Selected_Source_Code[L_i]);

    L_Fallback_Activated_Event :=
        L_Fallback_Active AND NOT L_Prev_Fallback_Active[L_i];

    L_Fallback_Recovered_Event :=
        (NOT L_Fallback_Active) AND L_Prev_Fallback_Active[L_i] AND NOT L_Source_Loss_Active;

    L_Source_Loss_Event :=
        L_Source_Loss_Active AND NOT L_Prev_Source_Loss[L_i];

    L_Last_Event_Code := 0;
    L_Last_Event_Text := '';

    IF L_Source_Loss_Event THEN
        L_Last_Event_Code := 4;
        L_Last_Event_Text := 'Temperature source loss';
    ELSIF L_Fallback_Activated_Event THEN
        L_Last_Event_Code := 2;
        L_Last_Event_Text := L_Reason_Text;
    ELSIF L_Fallback_Recovered_Event THEN
        L_Last_Event_Code := 3;
        L_Last_Event_Text := 'Fallback recovered; primary source selected';
    ELSIF L_Source_Switched_Event THEN
        L_Last_Event_Code := 1;
        L_Last_Event_Text := 'Temperature source switched';
    END_IF;

    GVL_Heating_Runtime_Projection.G_Circuit_Projection[L_i].Visible := TRUE;
    GVL_Heating_Runtime_Projection.G_Circuit_Projection[L_i].Selected_Source_Code := L_Selected_Source_Code;
    GVL_Heating_Runtime_Projection.G_Circuit_Projection[L_i].Selected_Source_Confidence := L_Selected_Confidence;
    GVL_Heating_Runtime_Projection.G_Circuit_Projection[L_i].Fallback_Active := L_Fallback_Active;
    GVL_Heating_Runtime_Projection.G_Circuit_Projection[L_i].Source_Degraded := L_Source_Degraded;
    GVL_Heating_Runtime_Projection.G_Circuit_Projection[L_i].Sensor_Error_Active := L_Sensor_Error;
    GVL_Heating_Runtime_Projection.G_Circuit_Projection[L_i].Reason_Code := L_Reason_Code;
    GVL_Heating_Runtime_Projection.G_Circuit_Projection[L_i].Reason_Text := L_Reason_Text;
    GVL_Heating_Runtime_Projection.G_Circuit_Projection[L_i].Source_Switched_Event := L_Source_Switched_Event;
    GVL_Heating_Runtime_Projection.G_Circuit_Projection[L_i].Fallback_Activated_Event := L_Fallback_Activated_Event;
    GVL_Heating_Runtime_Projection.G_Circuit_Projection[L_i].Fallback_Recovered_Event := L_Fallback_Recovered_Event;
    GVL_Heating_Runtime_Projection.G_Circuit_Projection[L_i].Source_Loss_Event := L_Source_Loss_Event;
    GVL_Heating_Runtime_Projection.G_Circuit_Projection[L_i].Last_Event_Code := L_Last_Event_Code;
    GVL_Heating_Runtime_Projection.G_Circuit_Projection[L_i].Last_Event_Text := L_Last_Event_Text;

    IF L_Last_Event_Code <> 0 THEN
        GVL_Heating_Runtime_Projection.G_Circuit_Projection[L_i].Last_Event_MS := VI_System_Time_MS;
    END_IF;

    L_Prev_Selected_Source_Code[L_i] := L_Selected_Source_Code;
    L_Prev_Fallback_Active[L_i] := L_Fallback_Active;
    L_Prev_Source_Loss[L_i] := L_Source_Loss_Active;

    IF L_Overheat_Timer[L_i].Q THEN
        VO_Zone_Valves[L_i] := FALSE;
    END_IF;

    FOR L_j := 1 TO GVL_CONSTANTS.C_MAX_RULES DO
        IF VI_Rule_Actions[L_j].Active AND VI_Rule_Actions[L_j].Target_ID = L_i THEN
            IF VI_Rule_Actions[L_j].Action_Type = E_Rule_Action_Type.ACTION_SET_FLOOR_HEATING THEN
                VO_Zone_Valves[L_i] := (VI_Rule_Actions[L_j].Value > REAL#0.5);
            END_IF;
        END_IF;
    END_FOR;
END_FOR;

// >>> BULK_SYNC_ANCHOR: FB_Heating_Circuit_Control <<<
END_FUNCTION_BLOCK

(* ---- FB_Heating_Manifold_Control.st ---- *)
// ==============================================================================
// Heating manifold control helper
// Internal refactoring helper for FB_Heating_System_Manager.
// Valve test override remains in FB_Heating_System_Manager for now.
// ==============================================================================
FUNCTION_BLOCK FB_Heating_Manifold_Control
VAR_INPUT
    VI_System_Time_MS : UDINT;
    VI_IsActivePLC : BOOL;
    VI_DHW_Heating_Demand : BOOL;
    VI_Freeze_Mode_Active : BOOL;
    VI_Target_Supply_Temp : REAL;
    VI_Any_Zone_Active : ARRAY[1..GVL_CONSTANTS.C_MAX_MANIFOLDS] OF BOOL;
END_VAR

VAR_IN_OUT
    VI_Manifold_Pressures : ARRAY[1..GVL_CONSTANTS.C_MAX_MANIFOLDS] OF REAL;
    VI_Manifold_Currents : ARRAY[1..GVL_CONSTANTS.C_MAX_MANIFOLDS] OF REAL;
    VI_Manifold_Temps_Supply : ARRAY[1..GVL_CONSTANTS.C_MAX_MANIFOLDS] OF REAL;
    VI_Manifold_Temps_Return : ARRAY[1..GVL_CONSTANTS.C_MAX_MANIFOLDS] OF REAL;
END_VAR

VAR_OUTPUT
    VO_Manifold_Pumps : ARRAY[1..GVL_CONSTANTS.C_MAX_MANIFOLDS] OF BOOL;
    VO_Manifold_Valves : ARRAY[1..GVL_CONSTANTS.C_MAX_MANIFOLDS] OF REAL;
    VO_Status : ARRAY[1..GVL_CONSTANTS.C_MAX_MANIFOLDS] OF ST_Manifold_Status;
END_VAR

VAR
    L_i : INT;
    L_Delta_T : REAL;
    L_PID_Valves : ARRAY[1..GVL_CONSTANTS.C_MAX_MANIFOLDS] OF FB_PID_Controller;
    L_PID_Timer : ARRAY[1..GVL_CONSTANTS.C_MAX_MANIFOLDS] OF FB_System_Timer;
    L_Pump_Run_Timer : ARRAY[1..GVL_CONSTANTS.C_MAX_MANIFOLDS] OF FB_System_Timer;
    L_Pump_Pause_Timer : ARRAY[1..GVL_CONSTANTS.C_MAX_MANIFOLDS] OF FB_System_Timer;
    L_Pump_In_Pause : ARRAY[1..GVL_CONSTANTS.C_MAX_MANIFOLDS] OF BOOL;
    L_Pump_Diag : ARRAY[1..GVL_CONSTANTS.C_MAX_MANIFOLDS] OF FB_Device_Predictive_Diag;
END_VAR

FOR L_i := 1 TO GVL_CONSTANTS.C_MAX_MANIFOLDS DO
    L_PID_Timer[L_i](IN := TRUE, PT := T#1s, VI_System_Time_MS := VI_System_Time_MS);
    IF L_PID_Timer[L_i].Q THEN
        L_PID_Timer[L_i](IN := FALSE, PT := T#1s, VI_System_Time_MS := VI_System_Time_MS);
        L_PID_Timer[L_i](IN := TRUE, PT := T#1s, VI_System_Time_MS := VI_System_Time_MS);

        L_PID_Valves[L_i](
            VI_SetPoint := VI_Target_Supply_Temp,
            VI_ProcessValue := VI_Manifold_Temps_Supply[L_i],
            VI_Kp := 2.0,
            VI_Tn := 120.0,
            VI_Tv := 0.0,
            VI_Y_Min := 0.0,
            VI_Y_Max := 100.0,
            VI_Cycle_Time_S := 1.0,
            VO_Output => VO_Manifold_Valves[L_i]
        );
    END_IF;

    L_Pump_Run_Timer[L_i](
        IN := VO_Manifold_Pumps[L_i] AND NOT L_Pump_In_Pause[L_i],
        PT := T#72h,
        VI_System_Time_MS := VI_System_Time_MS
    );
    IF L_Pump_Run_Timer[L_i].Q THEN
        L_Pump_In_Pause[L_i] := TRUE;
    END_IF;

    L_Pump_Pause_Timer[L_i](
        IN := L_Pump_In_Pause[L_i],
        PT := T#1h,
        VI_System_Time_MS := VI_System_Time_MS
    );
    IF L_Pump_Pause_Timer[L_i].Q THEN
        L_Pump_In_Pause[L_i] := FALSE;
    END_IF;

    IF VI_DHW_Heating_Demand THEN
        VO_Manifold_Pumps[L_i] := FALSE;
        VO_Manifold_Valves[L_i] := 0.0;
    ELSE
        VO_Manifold_Pumps[L_i] := VI_IsActivePLC AND VI_Any_Zone_Active[L_i] AND NOT L_Pump_In_Pause[L_i];
    END_IF;

    IF VI_Freeze_Mode_Active THEN
        VO_Manifold_Pumps[L_i] := TRUE;
        IF VO_Manifold_Valves[L_i] < 35.0 THEN
            VO_Manifold_Valves[L_i] := 35.0;
        END_IF;
    END_IF;

    VO_Status[L_i].Pump_On := VO_Manifold_Pumps[L_i];
    VO_Status[L_i].Pump_Current := VI_Manifold_Currents[L_i];
    VO_Status[L_i].Pressure := VI_Manifold_Pressures[L_i];
    VO_Status[L_i].Temp_Supply := VI_Manifold_Temps_Supply[L_i];
    VO_Status[L_i].Temp_Return := VI_Manifold_Temps_Return[L_i];
    VO_Status[L_i].Valve_Pos := VO_Manifold_Valves[L_i];

    L_Pump_Diag[L_i](
        VI_Current_Value := VI_Manifold_Currents[L_i],
        VI_Nominal_Value := 0.55,
        VI_Is_Running := VO_Manifold_Pumps[L_i],
        VI_Reset_Stats := FALSE,
        VI_System_Time_MS := VI_System_Time_MS,
        VIO_Health_Data := VO_Status[L_i].Health
    );

    IF VO_Manifold_Pumps[L_i] THEN
        L_Delta_T := VI_Manifold_Temps_Supply[L_i] - VI_Manifold_Temps_Return[L_i];

        VO_Status[L_i].Error := FALSE;
        VO_Status[L_i].Error_ID := 0;

        IF VI_Manifold_Currents[L_i] <= 0.01 THEN
            VO_Status[L_i].Error := TRUE;
            VO_Status[L_i].Error_ID := TO_WORD(GVL_CONFIG.ERR_PUMP_NO_CURRENT);
        ELSIF VI_Manifold_Currents[L_i] < 0.3 THEN
            VO_Status[L_i].Error := TRUE;
            VO_Status[L_i].Error_ID := TO_WORD(GVL_CONFIG.ERR_PUMP_UNDERCURRENT);
        ELSIF VI_Manifold_Currents[L_i] > 1.5 THEN
            VO_Status[L_i].Error := TRUE;
            VO_Status[L_i].Error_ID := TO_WORD(GVL_CONFIG.ERR_PUMP_OVERCURRENT);
        END_IF;

        IF (NOT VO_Status[L_i].Error) AND ((VI_Manifold_Pressures[L_i] < 1.5) OR (VI_Manifold_Pressures[L_i] > 2.5)) THEN
            VO_Status[L_i].Error := TRUE;
            VO_Status[L_i].Error_ID := TO_WORD(GVL_CONFIG.ERR_PRESSURE_OUT_OF_RANGE);
        END_IF;

        IF NOT VO_Status[L_i].Error THEN
            IF L_Delta_T < 5.0 THEN
                VO_Status[L_i].Error := TRUE;
                VO_Status[L_i].Error_ID := TO_WORD(GVL_CONFIG.ERR_DELTA_T_LOW);
            ELSIF L_Delta_T > 10.0 THEN
                VO_Status[L_i].Error := TRUE;
                VO_Status[L_i].Error_ID := TO_WORD(GVL_CONFIG.ERR_DELTA_T_HIGH);
            END_IF;
        END_IF;
    END_IF;
END_FOR;

// >>> BULK_SYNC_ANCHOR: FB_Heating_Manifold_Control <<<
END_FUNCTION_BLOCK

(* ---- FB_Heating_Output_Projection.st ---- *)
FUNCTION_BLOCK FB_Heating_Output_Projection
VAR_INPUT
    VI_Zone_Valves : ARRAY[1..GVL_CONSTANTS.C_MAX_HEATING_CIRCUITS] OF BOOL;
    VI_Manifold_Pumps : ARRAY[1..GVL_CONSTANTS.C_MAX_MANIFOLDS] OF BOOL;
    VI_Manifold_Valves : ARRAY[1..GVL_CONSTANTS.C_MAX_MANIFOLDS] OF REAL;
    VI_DHW_Heating_Pump : BOOL;
    VI_DHW_Circ_Pump : BOOL;
    VI_Backup_Circulation_Pump : BOOL;
    VI_Electric_Heater_Enable : BOOL;
END_VAR
VAR
    L_i : INT;
END_VAR

FOR L_i := 1 TO GVL_CONSTANTS.C_MAX_HEATING_CIRCUITS DO
    GVL_HEATING_OUTPUT.DO_Zone_Valves[L_i] := VI_Zone_Valves[L_i];
END_FOR;

FOR L_i := 1 TO GVL_CONSTANTS.C_MAX_MANIFOLDS DO
    GVL_HEATING_OUTPUT.DO_Manifold_Pumps[L_i] := VI_Manifold_Pumps[L_i];
    GVL_HEATING_OUTPUT.AO_Manifold_Valves[L_i] := REAL_TO_UINT(VI_Manifold_Valves[L_i] * 1000.0);
END_FOR;

GVL_HEATING_OUTPUT.DO_DHW_Heating_Pump := VI_DHW_Heating_Pump;
GVL_HEATING_OUTPUT.DO_DHW_Circ_Pump := VI_DHW_Circ_Pump;
GVL_HEATING_OUTPUT.DO_Backup_Circulation_Pump := VI_Backup_Circulation_Pump;
GVL_HEATING_OUTPUT.DO_Electric_Heater_Enable := VI_Electric_Heater_Enable;

END_FUNCTION_BLOCK
// >>> BULK_SYNC_ANCHOR: FB_Heating_Output_Projection <<<

(* ---- FB_Heating_Runtime_Service_Gating_Phase.st ---- *)
// ==============================================================================
// Heating runtime service gating phase
// Applies service/out-of-service and freeze hardware gating to computed outputs.
// Does NOT calculate heating demand and does NOT publish final state.
// ==============================================================================
FUNCTION_BLOCK FB_Heating_Runtime_Service_Gating_Phase
VAR_INPUT
    VI_Enable : BOOL;
END_VAR
VAR_IN_OUT
    VIO_Manifold_Pumps : ARRAY[1..GVL_CONSTANTS.C_MAX_MANIFOLDS] OF BOOL;
    VIO_Backup_Circulation_Pump : BOOL;
    VIO_Electric_Heater_Enable : BOOL;
    VIO_DHW_Heating_Pump : BOOL;
    VIO_DHW_Circ_Pump : BOOL;
    VIO_DHW_Status : ST_DHW_Status;
    VIO_Freeze_Risk_Status : BOOL;
END_VAR
VAR_OUTPUT
    VO_Executed : BOOL;
    VO_Valid : BOOL;
END_VAR
VAR
    L_i : INT;
END_VAR

VO_Executed := FALSE;
VO_Valid := FALSE;

IF NOT VI_Enable THEN
    RETURN;
END_IF;

GVL_STATUS.G_Diagnostics.Backup_Pump_Out_Of_Service := NOT GVL_CONFIG.G_Backup_Circulation_Pump_In_Service;
GVL_STATUS.G_Diagnostics.Electric_Heater_Out_Of_Service := NOT GVL_CONFIG.G_Electric_Heater_In_Service;

IF NOT GVL_CONFIG.G_Backup_Circulation_Pump_In_Service THEN
    VIO_Backup_Circulation_Pump := FALSE;
END_IF;

IF NOT GVL_CONFIG.G_Electric_Heater_In_Service THEN
    VIO_Electric_Heater_Enable := FALSE;
END_IF;

FOR L_i := 1 TO GVL_CONSTANTS.C_MAX_MANIFOLDS DO
    GVL_STATUS.G_Diagnostics.Manifold_Pump_Out_Of_Service[L_i] := NOT GVL_CONFIG.G_Manifold_Pump_In_Service[L_i];
    IF NOT GVL_CONFIG.G_Manifold_Pump_In_Service[L_i] THEN
        VIO_Manifold_Pumps[L_i] := FALSE;
    END_IF;
END_FOR;

GVL_STATUS.G_Diagnostics.DHW_Heating_Pump_Out_Of_Service := NOT GVL_CONFIG.G_DHW_Heating_Pump_In_Service;
IF NOT GVL_CONFIG.G_DHW_Heating_Pump_In_Service THEN
    VIO_DHW_Heating_Pump := FALSE;
    VIO_DHW_Status.Heating_Pump_On := FALSE;
END_IF;

GVL_STATUS.G_Diagnostics.DHW_Circ_Pump_Out_Of_Service := NOT GVL_CONFIG.G_DHW_Circ_Pump_In_Service;
IF NOT GVL_CONFIG.G_DHW_Circ_Pump_In_Service THEN
    VIO_DHW_Circ_Pump := FALSE;
    VIO_DHW_Status.Circ_Pump_On := FALSE;
END_IF;

GVL_STATE.G_Freeze_Hardware_Degraded := GVL_STATUS.G_Diagnostics.Backup_Pump_Fault OR GVL_STATUS.G_Diagnostics.Electric_Heater_Fault;
GVL_STATE.G_Freeze_Hardware_Failed := GVL_STATUS.G_Diagnostics.Backup_Pump_Fault AND GVL_STATUS.G_Diagnostics.Electric_Heater_Fault;

IF GVL_STATE.G_Freeze_Hardware_Failed THEN
    VIO_Backup_Circulation_Pump := FALSE;
    VIO_Electric_Heater_Enable := FALSE;
    VIO_Freeze_Risk_Status := TRUE;
END_IF;

VO_Executed := TRUE;
VO_Valid := TRUE;

END_FUNCTION_BLOCK
// >>> BULK_SYNC_ANCHOR: FB_Heating_Runtime_Service_Gating_Phase <<<

(* ---- FB_Heating_Runtime_Supervisory_Enrichment.st ---- *)
// ==============================================================================
// Heating runtime supervisory enrichment
// Passive observability-only connector for restored supervisory FB stack.
//
// DOES NOT own runtime.
// DOES NOT own heating logic.
// DOES NOT own diagnostics authority.
// DOES NOT own OpenTherm transport.
// DOES NOT write outputs or commands.
// ==============================================================================
FUNCTION_BLOCK FB_Heating_Runtime_Supervisory_Enrichment
VAR_INPUT
    VI_Enable : BOOL;
    VI_System_Time_MS : UDINT;
    VI_Runtime_Context : ST_Heating_Runtime_Context;
    VI_Phase_Event : ST_Heating_Runtime_Phase_Event;
    VI_Anomaly : ST_Heating_Runtime_Anomaly;
    VI_Cascade_Boiler_Count : UINT;
    VI_OT_Command_Valid : BOOL;
END_VAR
VAR_IN_OUT
    VIO_Event_Buffer : ST_Heating_Runtime_Event_Buffer;
    VIO_Execution_Timeline : ST_Heating_Runtime_Execution_Timeline;
END_VAR
VAR_OUTPUT
    VO_Causality_Node : ST_Heating_Runtime_Causality_Node;
    VO_Causality_Edge : ST_Heating_Runtime_Causality_Edge;
    VO_Blackbox_Event : ST_Heating_Runtime_Blackbox_Event;
    VO_Predictive_State : ST_Heating_Runtime_Predictive_State;
    VO_Status_Code : UINT;
    VO_Status_Text : STRING(128);
END_VAR
VAR
    fbEventManager : FB_Heating_Runtime_Event_Manager;
    fbTimelineObserver : FB_Heating_Runtime_Timeline_Observer;
    fbRootCauseCorrelator : FB_Heating_Runtime_RootCause_Correlator;
    fbReconstructionEngine : FB_Heating_Runtime_Event_Reconstruction_Engine;
    fbStabilityModel : FB_Heating_Runtime_Stability_Model;
    fbOTCascadeCorrelator : FB_Heating_Runtime_OT_Cascade_Correlator;
    fbOTInstabilityPredictor : FB_Heating_Runtime_OT_Instability_Predictor;
    fbPredictiveCorrelation : FB_Heating_Runtime_Predictive_Correlation_Weighting_Engine;

    L_Frame : ST_Heating_Runtime_Execution_Frame;
    L_Runtime_Risk : UINT;
    L_Cascade_Risk : UINT;
    L_Circuit_i : INT;
    L_Circuit_Event_Active : BOOL;
    L_Circuit_Event_Code : UINT;
    L_Circuit_Event_Text : STRING(128);
    L_Phase_Event : ST_Heating_Runtime_Phase_Event;
    L_Anomaly : ST_Heating_Runtime_Anomaly;

    L_Source_Instability_Max : REAL;
    L_Source_Instability_UINT : UINT;
    L_Source_Attention : BOOL;
    L_Source_Oscillation_Trend : BOOL;
    L_Source_Degraded_Trend : BOOL;
    L_Source_Loss_Trend : BOOL;
END_VAR

// ======================================================
// DEFAULTS
// ======================================================
VO_Status_Code := 0;
VO_Status_Text := 'Heating runtime supervisory enrichment disabled';

IF NOT VI_Enable THEN
    RETURN;
END_IF;

// ======================================================
// PASSIVE CIRCUIT EDGE INGESTION
// ======================================================
// Circuit control publishes canonical runtime projection only. This supervisory
// connector is the integration boundary that raises those passive projection
// edges into the event/anomaly stream used by timeline, reconstruction and
// causality observers.
L_Phase_Event := VI_Phase_Event;
L_Anomaly := VI_Anomaly;
L_Circuit_Event_Active := FALSE;
L_Circuit_Event_Code := 0;
L_Circuit_Event_Text := '';

FOR L_Circuit_i := 1 TO GVL_CONSTANTS.C_MAX_HEATING_CIRCUITS DO
    IF GVL_Heating_Runtime_Projection.G_Circuit_Projection[L_Circuit_i].Source_Loss_Event THEN
        L_Circuit_Event_Active := TRUE;
        L_Circuit_Event_Code := 804;
        L_Circuit_Event_Text := 'Heating circuit temperature source loss';
        EXIT;
    ELSIF GVL_Heating_Runtime_Projection.G_Circuit_Projection[L_Circuit_i].Fallback_Activated_Event THEN
        L_Circuit_Event_Active := TRUE;
        L_Circuit_Event_Code := 802;
        L_Circuit_Event_Text := 'Heating circuit fallback activated';
        EXIT;
    ELSIF GVL_Heating_Runtime_Projection.G_Circuit_Projection[L_Circuit_i].Fallback_Recovered_Event THEN
        L_Circuit_Event_Active := TRUE;
        L_Circuit_Event_Code := 803;
        L_Circuit_Event_Text := 'Heating circuit fallback recovered';
        EXIT;
    ELSIF GVL_Heating_Runtime_Projection.G_Circuit_Projection[L_Circuit_i].Source_Switched_Event THEN
        L_Circuit_Event_Active := TRUE;
        L_Circuit_Event_Code := 801;
        L_Circuit_Event_Text := 'Heating circuit temperature source switched';
        EXIT;
    END_IF;
END_FOR;

IF L_Circuit_Event_Active THEN
    L_Phase_Event.Phase := VI_Runtime_Context.Current_Phase;
    L_Phase_Event.Event_Active := TRUE;
    L_Phase_Event.Event_Completed := TRUE;
    L_Phase_Event.Event_Failed := FALSE;
    L_Phase_Event.Start_Time_MS := VI_System_Time_MS;
    L_Phase_Event.End_Time_MS := VI_System_Time_MS;
    L_Phase_Event.Duration_MS := 0;
    L_Phase_Event.Ordering_Valid := TRUE;
    L_Phase_Event.Isolation_Valid := TRUE;
    L_Phase_Event.Status_Code := L_Circuit_Event_Code;
    L_Phase_Event.Status_Text := L_Circuit_Event_Text;
    L_Phase_Event.Diagnostics_Visible := TRUE;
    L_Phase_Event.Explainability_Visible := TRUE;
    L_Phase_Event.Safety_Integrity_Valid := TRUE;
    L_Phase_Event.OpenTherm_Ownership_Valid := TRUE;
    L_Phase_Event.Cascade_Ownership_Valid := TRUE;

    L_Anomaly.Anomaly_Active := TRUE;
    L_Anomaly.Runtime_Degraded := L_Anomaly.Runtime_Degraded OR (L_Circuit_Event_Code = 802) OR (L_Circuit_Event_Code = 804);
    L_Anomaly.Diagnostics_Degraded := L_Anomaly.Diagnostics_Degraded OR (L_Circuit_Event_Code = 804);
    L_Anomaly.Explainability_Degraded := L_Anomaly.Explainability_Degraded OR (L_Circuit_Event_Code = 804);

    IF L_Circuit_Event_Code = 804 THEN
        IF L_Anomaly.Severity_Level < 80 THEN
            L_Anomaly.Severity_Level := 80;
        END_IF;
        L_Anomaly.Status_Code := 804;
        L_Anomaly.Status_Text := 'Heating circuit source loss observed';
    ELSIF L_Circuit_Event_Code = 802 THEN
        IF L_Anomaly.Severity_Level < 40 THEN
            L_Anomaly.Severity_Level := 40;
        END_IF;
        L_Anomaly.Status_Code := 802;
        L_Anomaly.Status_Text := 'Heating circuit fallback activation observed';
    ELSIF L_Circuit_Event_Code = 803 THEN
        L_Anomaly.Status_Code := 803;
        L_Anomaly.Status_Text := 'Heating circuit fallback recovery observed';
    ELSE
        L_Anomaly.Status_Code := 801;
        L_Anomaly.Status_Text := 'Heating circuit source switch observed';
    END_IF;
END_IF;

// ======================================================
// SOURCE INSTABILITY AGGREGATION
// ======================================================
// Per-circuit predictive details remain in GVL_Heating_Source_Stability.G_State.
// This supervisory layer publishes only the aggregate source-instability view
// into the canonical runtime predictive state.
L_Source_Instability_Max := REAL#0.0;
L_Source_Attention := FALSE;
L_Source_Oscillation_Trend := FALSE;
L_Source_Degraded_Trend := FALSE;
L_Source_Loss_Trend := FALSE;

FOR L_Circuit_i := 1 TO GVL_CONSTANTS.C_MAX_HEATING_CIRCUITS DO
    IF GVL_Heating_Source_Stability.G_State[L_Circuit_i].Instability_Score > L_Source_Instability_Max THEN
        L_Source_Instability_Max := GVL_Heating_Source_Stability.G_State[L_Circuit_i].Instability_Score;
    END_IF;

    L_Source_Attention :=
        L_Source_Attention OR
        GVL_Heating_Source_Stability.G_State[L_Circuit_i].Instability_Attention;

    L_Source_Oscillation_Trend :=
        L_Source_Oscillation_Trend OR
        GVL_Heating_Source_Stability.G_State[L_Circuit_i].Oscillation_Detected;

    L_Source_Degraded_Trend :=
        L_Source_Degraded_Trend OR
        GVL_Heating_Source_Stability.G_State[L_Circuit_i].Degraded_Trend_Visible;

    L_Source_Loss_Trend :=
        L_Source_Loss_Trend OR
        (GVL_Heating_Source_Stability.G_State[L_Circuit_i].Source_Loss_Count > 0);
END_FOR;

IF L_Source_Instability_Max < REAL#0.0 THEN
    L_Source_Instability_UINT := 0;
ELSIF L_Source_Instability_Max > REAL#100.0 THEN
    L_Source_Instability_UINT := 100;
ELSE
    L_Source_Instability_UINT := REAL_TO_UINT(L_Source_Instability_Max);
END_IF;

// ======================================================
// EXECUTION FRAME FROM CURRENT RUNTIME CONTEXT
// ======================================================
L_Frame.Phase := VI_Runtime_Context.Current_Phase;
L_Frame.Frame_Started := TRUE;
L_Frame.Frame_Completed := VI_Runtime_Context.Output_Projection_Executed;
L_Frame.Frame_Failed := VI_Runtime_Context.Runtime_Fault;
L_Frame.Frame_Start_MS := VI_System_Time_MS;
L_Frame.Frame_End_MS := VI_System_Time_MS;
L_Frame.Frame_Duration_MS := 0;

L_Frame.Sequencing_Valid :=
    VI_Runtime_Context.DHW_Before_Heating_Valid AND
    VI_Runtime_Context.State_Publication_Before_Diagnostics_Valid AND
    VI_Runtime_Context.Output_Projection_Last_Valid;

L_Frame.Ownership_Valid :=
    VI_Runtime_Context.OpenTherm_Ownership_Valid AND
    VI_Runtime_Context.Cascade_Ownership_Valid AND
    VI_Runtime_Context.Safety_Isolation_Valid;

L_Frame.Synchronization_Valid :=
    VI_Runtime_Context.Diagnostics_Isolation_Valid AND
    VI_Runtime_Context.Explainability_Isolation_Valid;

L_Frame.Runtime_Jitter_Detected := L_Anomaly.Runtime_Jitter_Detected;
L_Frame.Runtime_Latency_Detected := L_Anomaly.Runtime_Latency_Detected;
L_Frame.Runtime_Degraded := L_Anomaly.Runtime_Degraded;
L_Frame.Status_Code := VI_Runtime_Context.Runtime_Status_Code;
L_Frame.Status_Text := VI_Runtime_Context.Runtime_Status_Text;

fbTimelineObserver(
    VI_Enable := TRUE,
    VI_Frame := L_Frame,
    VIO_Timeline := VIO_Execution_Timeline
);

// ======================================================
// EVENT BUFFER
// ======================================================
fbEventManager(
    VI_Enable := TRUE,
    VI_Event := L_Phase_Event,
    VIO_Buffer := VIO_Event_Buffer
);

// ======================================================
// ROOT-CAUSE / CAUSALITY NODE
// ======================================================
fbRootCauseCorrelator(
    VI_Enable := TRUE,
    VI_Anomaly := L_Anomaly
);

VO_Causality_Node := fbRootCauseCorrelator.VO_Node;

// ======================================================
// CAUSALITY EDGE BUILT FROM NODE STATE
// ======================================================
VO_Causality_Edge.Source_Node_ID := 1;
VO_Causality_Edge.Target_Node_ID := 2;
VO_Causality_Edge.Edge_Active := VO_Causality_Node.Node_Active;
VO_Causality_Edge.Propagation_Detected :=
    VO_Causality_Node.Runtime_Degraded OR
    VO_Causality_Node.Runtime_Fault OR
    VO_Causality_Node.Cascade_Degraded OR
    VO_Causality_Node.OpenTherm_Degraded OR
    VO_Causality_Node.Sequencing_Invalid OR
    VO_Causality_Node.Ownership_Invalid OR
    VO_Causality_Node.Synchronization_Invalid;

VO_Causality_Edge.Runtime_Propagation :=
    VO_Causality_Node.Runtime_Degraded OR VO_Causality_Node.Runtime_Fault;
VO_Causality_Edge.Cascade_Propagation := VO_Causality_Node.Cascade_Degraded;
VO_Causality_Edge.OpenTherm_Propagation := VO_Causality_Node.OpenTherm_Degraded;
VO_Causality_Edge.Diagnostics_Propagation := VO_Causality_Node.Diagnostics_Degraded;
VO_Causality_Edge.Sequencing_Propagation := VO_Causality_Node.Sequencing_Invalid;
VO_Causality_Edge.Ownership_Propagation := VO_Causality_Node.Ownership_Invalid;
VO_Causality_Edge.Synchronization_Propagation := VO_Causality_Node.Synchronization_Invalid;
VO_Causality_Edge.Severity_Level := VO_Causality_Node.Severity_Level;
VO_Causality_Edge.Critical_Path := VO_Causality_Node.Root_Cause_Candidate;
VO_Causality_Edge.Status_Code := VO_Causality_Node.Status_Code;
VO_Causality_Edge.Status_Text := VO_Causality_Node.Status_Text;

// ======================================================
// FORENSIC RECONSTRUCTION
// ======================================================
fbReconstructionEngine(
    VI_Enable := TRUE,
    VI_Node := VO_Causality_Node,
    VI_Edge := VO_Causality_Edge,
    VI_System_Time_MS := VI_System_Time_MS
);

VO_Blackbox_Event := fbReconstructionEngine.VO_Event;

// ======================================================
// STABILITY / OT / CASCADE PREDICTIVE SUPERVISION
// ======================================================
fbStabilityModel(
    VI_Enable := TRUE,
    VI_Runtime_Degraded := L_Anomaly.Runtime_Degraded,
    VI_Runtime_Critical := L_Anomaly.Critical_Anomaly
);

fbOTCascadeCorrelator(
    VI_Enable := TRUE,
    VI_Cascade_Degraded := L_Anomaly.Cascade_Degraded,
    VI_OT_Degraded := L_Anomaly.OpenTherm_Transport_Degraded,
    VI_OT_Command_Valid := VI_OT_Command_Valid,
    VI_Boiler_Count := VI_Cascade_Boiler_Count
);

fbOTInstabilityPredictor(
    VI_Enable := TRUE,
    VI_OT_Degraded := L_Anomaly.OpenTherm_Transport_Degraded,
    VI_OT_Command_Valid := VI_OT_Command_Valid
);

IF L_Anomaly.Critical_Anomaly THEN
    L_Runtime_Risk := 100;
ELSIF L_Anomaly.Runtime_Degraded THEN
    L_Runtime_Risk := 60;
ELSE
    L_Runtime_Risk := 0;
END_IF;

IF L_Anomaly.Cascade_Boiler_Loss_Detected THEN
    L_Cascade_Risk := 100;
ELSIF L_Anomaly.Cascade_Degraded THEN
    L_Cascade_Risk := 60;
ELSE
    L_Cascade_Risk := 0;
END_IF;

fbPredictiveCorrelation(
    VI_Enable := TRUE,
    VI_Runtime_Risk := L_Runtime_Risk,
    VI_Cascade_Risk := L_Cascade_Risk,
    VI_OT_Risk := fbOTInstabilityPredictor.VO_OT_Instability_Risk
);

// ======================================================
// PREDICTIVE PUBLICATION MODEL
// ======================================================
VO_Predictive_State.Predictive_Analytics_Visible := TRUE;
VO_Predictive_State.Predictive_Analytics_Degraded :=
    fbPredictiveCorrelation.VO_Correlation_Degraded OR L_Source_Attention;
VO_Predictive_State.Predictive_Analytics_Attention :=
    (fbPredictiveCorrelation.VO_Correlation_Score > 40) OR L_Source_Attention;
VO_Predictive_State.Runtime_Stable := fbStabilityModel.VO_Runtime_Stable;
VO_Predictive_State.Runtime_Stability_Score := fbStabilityModel.VO_Stability_Score;
VO_Predictive_State.Runtime_Degradation_Observation := L_Runtime_Risk;
VO_Predictive_State.Runtime_Failure_Observation := SEL(L_Anomaly.Critical_Anomaly, 0, 100);
VO_Predictive_State.Source_Instability_Observation := L_Source_Instability_UINT;
VO_Predictive_State.Source_Instability_Attention := L_Source_Attention;
VO_Predictive_State.Source_Oscillation_Trend_Visible := L_Source_Oscillation_Trend;
VO_Predictive_State.Source_Degraded_Trend_Visible := L_Source_Degraded_Trend;
VO_Predictive_State.Source_Loss_Trend_Visible := L_Source_Loss_Trend;
VO_Predictive_State.Cascade_Degradation_Observation := L_Cascade_Risk;
VO_Predictive_State.Cascade_Degraded_Trend_Visible := fbOTCascadeCorrelator.VO_Correlation_Detected;
VO_Predictive_State.OpenTherm_Instability_Observation := fbOTInstabilityPredictor.VO_OT_Instability_Risk;
VO_Predictive_State.OpenTherm_Degraded_Trend_Visible := fbOTInstabilityPredictor.VO_OT_Degraded_Trend;
VO_Predictive_State.Sequencing_Observation := SEL(VO_Causality_Node.Sequencing_Invalid, 0, 100);
VO_Predictive_State.Ownership_Observation := SEL(VO_Causality_Node.Ownership_Invalid, 0, 100);
VO_Predictive_State.Synchronization_Observation := SEL(VO_Causality_Node.Synchronization_Invalid, 0, 100);
VO_Predictive_State.Status_Code := fbPredictiveCorrelation.VO_Status_Code;

IF L_Source_Attention THEN
    VO_Predictive_State.Status_Text := 'Predictive analytics attention: heating source instability observed';
ELSE
    VO_Predictive_State.Status_Text := fbPredictiveCorrelation.VO_Status_Text;
END_IF;

VO_Status_Code := VO_Predictive_State.Status_Code;
VO_Status_Text := VO_Predictive_State.Status_Text;

END_FUNCTION_BLOCK
// >>> BULK_SYNC_ANCHOR: FB_Heating_Runtime_Supervisory_Enrichment <<<
